LIN {X 0,Y 404.214,Z 398.218,A -85,B 0,C 180,E1 -10998.599,E2 -10998.599} C_VEL
LIN {X 0,Y 404.141,Z 398.144,A -85,B 0,C 180,E1 -11001.419,E2 -11001.419} C_VEL
LIN {X 0,Y 404.175,Z 398.142,A -85,B 0,C 180,E1 -11004.666,E2 -11004.666} C_VEL
LIN {X 0,Y 404.133,Z 398.136,A -85,B 0,C 180,E1 -11008.005,E2 -11008.005} C_VEL
LIN {X 0,Y 404.147,Z 398.137,A -85,B 0,C 180,E1 -11010.285,E2 -11010.285} C_VEL
LIN {X 0,Y 404.146,Z 398.13,A -85,B 0,C 180,E1 -11013.812,E2 -11013.812} C_VEL
LIN {X 0,Y 404.138,Z 398.142,A -85,B 0,C 180,E1 -11016.875,E2 -11016.875} C_VEL
LIN {X 0,Y 404.149,Z 398.142,A -85,B 0,C 180,E1 -11020.08,E2 -11020.08} C_VEL
LIN {X 0,Y 404.152,Z 398.144,A -85,B 0,C 180,E1 -11023.083,E2 -11023.083} C_VEL
LIN {X 0,Y 404.149,Z 398.138,A -85,B 0,C 180,E1 -11025.926,E2 -11025.926} C_VEL
LIN {X 0,Y 404.115,Z 398.146,A -85,B 0,C 180,E1 -11028.634,E2 -11028.634} C_VEL
LIN {X 0,Y 404.143,Z 398.126,A -85,B 0,C 180,E1 -11031.495,E2 -11031.495} C_VEL
LIN {X 0,Y 404.186,Z 398.126,A -85,B 0,C 180,E1 -11034.984,E2 -11034.984} C_VEL
LIN {X 0,Y 404.205,Z 398.311,A -85,B 0,C 180,E1 -11037.017,E2 -11037.017} C_VEL
LIN {X 0,Y 408.291,Z 414.179,A -85,B 0,C 180,E1 -11039.741,E2 -11039.741} C_VEL
LIN {X 0,Y 410.43,Z 423.971,A -85,B 0,C 180,E1 -11041.35,E2 -11041.35} C_VEL
LIN {X 0,Y 409.654,Z 440.641,A -85,B 0,C 180,E1 -11043.783,E2 -11043.783} C_VEL
LIN {X 0,Y 408.396,Z 462.743,A -85,B 0,C 180,E1 -11046.952,E2 -11046.952} C_VEL
LIN {X 0,Y 407.404,Z 484.784,A -85,B 0,C 180,E1 -11049.962,E2 -11049.962} C_VEL
LIN {X 0,Y 407.308,Z 487.804,A -85,B 0,C 180,E1 -11050.352,E2 -11050.352} C_VEL
LIN {X 0,Y 410.444,Z 509.789,A -85,B 0,C 180,E1 -11050.926,E2 -11050.926} C_VEL
LIN {X 0,Y 409.306,Z 600.036,A -85,B 0,C 180,E1 -11052.546,E2 -11052.546} C_VEL
LIN {X 0,Y 408.805,Z 613.109,A -85,B 0,C 180,E1 -11052.975,E2 -11052.975} C_VEL
LIN {X 0,Y 408.172,Z 626.084,A -85,B 0,C 180,E1 -11053.623,E2 -11053.623} C_VEL
LIN {X 0,Y 407.355,Z 638.791,A -85,B 0,C 180,E1 -11054.489,E2 -11054.489} C_VEL
LIN {X 0,Y 407.145,Z 642.093,A -85,B 0,C 180,E1 -11054.761,E2 -11054.761} C_VEL
LIN {X 0,Y 406.21,Z 647.1,A -85,B 0,C 180,E1 -11055.184,E2 -11055.184} C_VEL
LIN {X 0,Y 402.866,Z 654.993,A -85,B 0,C 180,E1 -11055.892,E2 -11055.892} C_VEL
LIN {X 0,Y 399.431,Z 662.416,A -85,B 0,C 180,E1 -11056.697,E2 -11056.697} C_VEL
LIN {X 0,Y 398.364,Z 666.666,A -85,B 0,C 180,E1 -11057.267,E2 -11057.267} C_VEL
LIN {X 0,Y 397.512,Z 676.011,A -85,B 0,C 180,E1 -11058.786,E2 -11058.786} C_VEL
LIN {X 0,Y 396.894,Z 683.473,A -85,B 0,C 180,E1 -11060.316,E2 -11060.316} C_VEL
LIN {X 0,Y 396.405,Z 689.464,A -85,B 0,C 180,E1 -11061.846,E2 -11061.846} C_VEL
LIN {X 0,Y 396.121,Z 694.52,A -85,B 0,C 180,E1 -11063.493,E2 -11063.493} C_VEL
LIN {X 0,Y 395.956,Z 697.833,A -85,B 0,C 180,E1 -11064.909,E2 -11064.909} C_VEL
LIN {X 0,Y 395.809,Z 699.703,A -85,B 0,C 180,E1 -11065.927,E2 -11065.927} C_VEL
LIN {X 0,Y 395.742,Z 701.131,A -85,B 0,C 180,E1 -11066.946,E2 -11066.946} C_VEL
LIN {X 0,Y 395.764,Z 702.132,A -85,B 0,C 180,E1 -11067.965,E2 -11067.965} C_VEL
LIN {X 0,Y 395.76,Z 702.986,A -85,B 0,C 180,E1 -11070,E2 -11070} C_VEL
LIN {X 0,Y 395.76,Z 702.794,A -85,B 0,C 180,E1 -11071.018,E2 -11071.018} C_VEL
LIN {X 0,Y 395.764,Z 702.205,A -85,B 0,C 180,E1 -11072.036,E2 -11072.036} C_VEL
LIN {X 0,Y 395.808,Z 699.863,A -85,B 0,C 180,E1 -11074.073,E2 -11074.073} C_VEL
LIN {X 0,Y 395.992,Z 696.979,A -85,B 0,C 180,E1 -11075.602,E2 -11075.602} C_VEL
LIN {X 0,Y 396.133,Z 693.063,A -85,B 0,C 180,E1 -11077.134,E2 -11077.134} C_VEL
LIN {X 0,Y 396.528,Z 687.99,A -85,B 0,C 180,E1 -11078.665,E2 -11078.665} C_VEL
LIN {X 0,Y 397.018,Z 681.596,A -85,B 0,C 180,E1 -11080.196,E2 -11080.196} C_VEL
LIN {X 0,Y 397.716,Z 673.654,A -85,B 0,C 180,E1 -11081.725,E2 -11081.725} C_VEL
LIN {X 0,Y 398.485,Z 665.541,A -85,B 0,C 180,E1 -11082.995,E2 -11082.995} C_VEL
LIN {X 0,Y 399.348,Z 655.573,A -85,B 0,C 180,E1 -11084.264,E2 -11084.264} C_VEL
LIN {X 0,Y 400.006,Z 645.746,A -85,B 0,C 180,E1 -11085.281,E2 -11085.281} C_VEL
LIN {X 0,Y 400.808,Z 635.099,A -85,B 0,C 180,E1 -11086.163,E2 -11086.163} C_VEL
LIN {X 0,Y 401.56,Z 623.437,A -85,B 0,C 180,E1 -11086.916,E2 -11086.916} C_VEL
LIN {X 0,Y 402.197,Z 610.726,A -85,B 0,C 180,E1 -11087.511,E2 -11087.511} C_VEL
LIN {X 0,Y 402.613,Z 597.392,A -85,B 0,C 180,E1 -11087.919,E2 -11087.919} C_VEL
LIN {X 0,Y 403.64,Z 509.348,A -85,B 0,C 180,E1 -11089.513,E2 -11089.513} C_VEL
LIN {X 0,Y 400.563,Z 487.69,A -85,B 0,C 180,E1 -11090.101,E2 -11090.101} C_VEL
LIN {X 0,Y 401.538,Z 465.188,A -85,B 0,C 180,E1 -11093.192,E2 -11093.192} C_VEL
LIN {X 0,Y 403.073,Z 439.157,A -85,B 0,C 180,E1 -11096.958,E2 -11096.958} C_VEL
LIN {X 0,Y 403.764,Z 426.144,A -85,B 0,C 180,E1 -11098.883,E2 -11098.883} C_VEL
LIN {X 0,Y 400.633,Z 412.28,A -85,B 0,C 180,E1 -11101.2,E2 -11101.2} C_VEL
LIN {X 0,Y 397.148,Z 399.203,A -85,B 0,C 180,E1 -11103.492,E2 -11103.492} C_VEL
LIN {X 0,Y 397.096,Z 399.012,A -85,B 0,C 180,E1 -11106.996,E2 -11106.996} C_VEL
LIN {X 0,Y 397.057,Z 399.012,A -85,B 0,C 180,E1 -11110.438,E2 -11110.438} C_VEL
LIN {X 0,Y 397.089,Z 399.01,A -85,B 0,C 180,E1 -11113.651,E2 -11113.651} C_VEL
LIN {X 0,Y 397.101,Z 399.019,A -85,B 0,C 180,E1 -11116.522,E2 -11116.522} C_VEL
LIN {X 0,Y 397.088,Z 399.022,A -85,B 0,C 180,E1 -11120.42,E2 -11120.42} C_VEL
LIN {X 0,Y 397.097,Z 399.012,A -85,B 0,C 180,E1 -11123.005,E2 -11123.005} C_VEL
LIN {X 0,Y 397.115,Z 399.006,A -85,B 0,C 180,E1 -11126.727,E2 -11126.727} C_VEL
LIN {X 0,Y 397.12,Z 399.011,A -85,B 0,C 180,E1 -11130.295,E2 -11130.295} C_VEL
LIN {X 0,Y 397.08,Z 399.027,A -85,B 0,C 180,E1 -11133.738,E2 -11133.738} C_VEL
LIN {X 0,Y 397.102,Z 399.008,A -85,B 0,C 180,E1 -11137.085,E2 -11137.085} C_VEL
LIN {X 0,Y 397.149,Z 399.009,A -85,B 0,C 180,E1 -11140.353,E2 -11140.353} C_VEL
LIN {X 0,Y 397.132,Z 399.008,A -85,B 0,C 180,E1 -11143.552,E2 -11143.552} C_VEL
LIN {X 0,Y 397.233,Z 398.998,A -85,B 0,C 180,E1 -11146.703,E2 -11146.703} C_VEL
LIN {X 0,Y 397.209,Z 398.996,A -85,B 0,C 180,E1 -11149.809,E2 -11149.809} C_VEL
LIN {X 0,Y 397.297,Z 398.992,A -85,B 0,C 180,E1 -11152.887,E2 -11152.887} C_VEL
LIN {X 0,Y 397.231,Z 398.989,A -85,B 0,C 180,E1 -11154.925,E2 -11154.925} C_VEL
LIN {X 0,Y 397.443,Z 398.978,A -85,B 0,C 180,E1 -11157.973,E2 -11157.973} C_VEL
LIN {X 0,Y 397.442,Z 398.959,A -85,B 0,C 180,E1 -11162.027,E2 -11162.027} C_VEL
LIN {X 0,Y 397.331,Z 398.992,A -85,B 0,C 180,E1 -11166.092,E2 -11166.092} C_VEL
LIN {X 0,Y 397.23,Z 398.989,A -85,B 0,C 180,E1 -11169.162,E2 -11169.162} C_VEL
LIN {X 0,Y 397.217,Z 399.005,A -85,B 0,C 180,E1 -11172.258,E2 -11172.258} C_VEL
LIN {X 0,Y 397.113,Z 399.01,A -85,B 0,C 180,E1 -11175.395,E2 -11175.395} C_VEL
LIN {X 0,Y 397.084,Z 399.018,A -85,B 0,C 180,E1 -11178.577,E2 -11178.577} C_VEL
LIN {X 0,Y 397.091,Z 399.012,A -85,B 0,C 180,E1 -11181.819,E2 -11181.819} C_VEL
LIN {X 0,Y 397.104,Z 399.015,A -85,B 0,C 180,E1 -11185.135,E2 -11185.135} C_VEL
LIN {X 0,Y 397.064,Z 399.01,A -85,B 0,C 180,E1 -11188.548,E2 -11188.548} C_VEL
LIN {X 0,Y 397.083,Z 399.026,A -85,B 0,C 180,E1 -11191.836,E2 -11191.836} C_VEL
LIN {X 0,Y 397.119,Z 399.007,A -85,B 0,C 180,E1 -11194.494,E2 -11194.494} C_VEL
LIN {X 0,Y 397.088,Z 399.015,A -85,B 0,C 180,E1 -11198.277,E2 -11198.277} C_VEL
LIN {X 0,Y 397.051,Z 398.989,A -85,B 0,C 180,E1 -11201.976,E2 -11201.976} C_VEL
LIN {X 0,Y 397.085,Z 399.02,A -85,B 0,C 180,E1 -11205.069,E2 -11205.069} C_VEL
LIN {X 0,Y 397.051,Z 398.999,A -85,B 0,C 180,E1 -11208.024,E2 -11208.024} C_VEL
LIN {X 0,Y 397.089,Z 399.017,A -85,B 0,C 180,E1 -11211.146,E2 -11211.146} C_VEL
LIN {X 0,Y 397.098,Z 399.022,A -85,B 0,C 180,E1 -11214.501,E2 -11214.501} C_VEL
LIN {X 0,Y 397.186,Z 399.276,A -85,B 0,C 180,E1 -11216.827,E2 -11216.827} C_VEL
LIN {X 0,Y 401.583,Z 418.852,A -85,B 0,C 180,E1 -11220.37,E2 -11220.37} C_VEL
LIN {X 0,Y 402.413,Z 422.758,A -85,B 0,C 180,E1 -11221.052,E2 -11221.052} C_VEL
LIN {X 0,Y 401.237,Z 439.938,A -85,B 0,C 180,E1 -11223.795,E2 -11223.795} C_VEL
LIN {X 0,Y 399.68,Z 461.77,A -85,B 0,C 180,E1 -11227.241,E2 -11227.241} C_VEL
LIN {X 0,Y 398.867,Z 475.69,A -85,B 0,C 180,E1 -11229.399,E2 -11229.399} C_VEL
LIN {X 0,Y 399.784,Z 488.481,A -85,B 0,C 180,E1 -11230.077,E2 -11230.077} C_VEL
LIN {X 0,Y 403.137,Z 518.848,A -85,B 0,C 180,E1 -11230.811,E2 -11230.811} C_VEL
LIN {X 0,Y 402.076,Z 606.296,A -85,B 0,C 180,E1 -11232.385,E2 -11232.385} C_VEL
LIN {X 0,Y 401.5,Z 619.645,A -85,B 0,C 180,E1 -11232.819,E2 -11232.819} C_VEL
LIN {X 0,Y 400.956,Z 632.32,A -85,B 0,C 180,E1 -11233.451,E2 -11233.451} C_VEL
LIN {X 0,Y 400.243,Z 643.58,A -85,B 0,C 180,E1 -11234.206,E2 -11234.206} C_VEL
LIN {X 0,Y 399.446,Z 654.245,A -85,B 0,C 180,E1 -11235.128,E2 -11235.128} C_VEL
LIN {X 0,Y 398.711,Z 664.528,A -85,B 0,C 180,E1 -11236.242,E2 -11236.242} C_VEL
LIN {X 0,Y 397.975,Z 673.995,A -85,B 0,C 180,E1 -11237.506,E2 -11237.506} C_VEL
LIN {X 0,Y 397.237,Z 681.776,A -85,B 0,C 180,E1 -11238.778,E2 -11238.778} C_VEL
LIN {X 0,Y 396.694,Z 689.349,A -85,B 0,C 180,E1 -11240.31,E2 -11240.31} C_VEL
LIN {X 0,Y 396.282,Z 695.425,A -85,B 0,C 180,E1 -11241.843,E2 -11241.843} C_VEL
LIN {X 0,Y 396.022,Z 700.221,A -85,B 0,C 180,E1 -11243.376,E2 -11243.376} C_VEL
LIN {X 0,Y 395.955,Z 703.879,A -85,B 0,C 180,E1 -11244.908,E2 -11244.908} C_VEL
LIN {X 0,Y 395.846,Z 705.763,A -85,B 0,C 180,E1 -11245.927,E2 -11245.927} C_VEL
LIN {X 0,Y 395.804,Z 707.185,A -85,B 0,C 180,E1 -11246.946,E2 -11246.946} C_VEL
LIN {X 0,Y 395.844,Z 708.188,A -85,B 0,C 180,E1 -11247.965,E2 -11247.965} C_VEL
LIN {X 0,Y 395.832,Z 708.801,A -85,B 0,C 180,E1 -11248.983,E2 -11248.983} C_VEL
LIN {X 0,Y 395.828,Z 709.02,A -85,B 0,C 180,E1 -11250,E2 -11250} C_VEL
LIN {X 0,Y 395.857,Z 708.799,A -85,B 0,C 180,E1 -11251.017,E2 -11251.017} C_VEL
LIN {X 0,Y 395.848,Z 708.184,A -85,B 0,C 180,E1 -11252.035,E2 -11252.035} C_VEL
LIN {X 0,Y 395.811,Z 707.18,A -85,B 0,C 180,E1 -11253.053,E2 -11253.053} C_VEL
LIN {X 0,Y 395.855,Z 705.755,A -85,B 0,C 180,E1 -11254.072,E2 -11254.072} C_VEL
LIN {X 0,Y 395.967,Z 702.789,A -85,B 0,C 180,E1 -11255.602,E2 -11255.602} C_VEL
LIN {X 0,Y 396.102,Z 698.758,A -85,B 0,C 180,E1 -11257.134,E2 -11257.134} C_VEL
LIN {X 0,Y 396.525,Z 692.538,A -85,B 0,C 180,E1 -11258.922,E2 -11258.922} C_VEL
LIN {X 0,Y 396.98,Z 685.747,A -85,B 0,C 180,E1 -11260.455,E2 -11260.455} C_VEL
LIN {X 0,Y 397.539,Z 678.792,A -85,B 0,C 180,E1 -11261.73,E2 -11261.73} C_VEL
LIN {X 0,Y 398.233,Z 670.382,A -85,B 0,C 180,E1 -11263.003,E2 -11263.003} C_VEL
LIN {X 0,Y 399.039,Z 659.963,A -85,B 0,C 180,E1 -11264.275,E2 -11264.275} C_VEL
LIN {X 0,Y 399.789,Z 649.629,A -85,B 0,C 180,E1 -11265.289,E2 -11265.289} C_VEL
LIN {X 0,Y 400.544,Z 638.228,A -85,B 0,C 180,E1 -11266.173,E2 -11266.173} C_VEL
LIN {X 0,Y 401.28,Z 626.381,A -85,B 0,C 180,E1 -11266.862,E2 -11266.862} C_VEL
LIN {X 0,Y 401.815,Z 613.578,A -85,B 0,C 180,E1 -11267.396,E2 -11267.396} C_VEL
LIN {X 0,Y 402.155,Z 599.896,A -85,B 0,C 180,E1 -11267.742,E2 -11267.742} C_VEL
LIN {X 0,Y 402.409,Z 587.532,A -85,B 0,C 180,E1 -11267.993,E2 -11267.993} C_VEL
LIN {X 0,Y 403.421,Z 551.708,A -85,B 0,C 180,E1 -11268.867,E2 -11268.867} C_VEL
LIN {X 0,Y 404.277,Z 517.801,A -85,B 0,C 180,E1 -11269.699,E2 -11269.699} C_VEL
LIN {X 0,Y 402.318,Z 492.103,A -85,B 0,C 180,E1 -11270.547,E2 -11270.547} C_VEL
LIN {X 0,Y 399.514,Z 472.889,A -85,B 0,C 180,E1 -11271.317,E2 -11271.317} C_VEL
LIN {X 0,Y 399.185,Z 470.402,A -85,B 0,C 180,E1 -11271.458,E2 -11271.458} C_VEL
LIN {X 0,Y 400.855,Z 449.87,A -85,B 0,C 180,E1 -11274.884,E2 -11274.884} C_VEL
LIN {X 0,Y 402.767,Z 431.494,A -85,B 0,C 180,E1 -11278.108,E2 -11278.108} C_VEL
LIN {X 0,Y 403.442,Z 425.577,A -85,B 0,C 180,E1 -11279.194,E2 -11279.194} C_VEL
LIN {X 0,Y 402.201,Z 418.214,A -85,B 0,C 180,E1 -11280.782,E2 -11280.782} C_VEL
LIN {X 0,Y 399.687,Z 407.941,A -85,B 0,C 180,E1 -11283.271,E2 -11283.271} C_VEL
LIN {X 0,Y 397.125,Z 399.276,A -85,B 0,C 180,E1 -11285.733,E2 -11285.733} C_VEL
LIN {X 0,Y 397.087,Z 399.023,A -85,B 0,C 180,E1 -11287.207,E2 -11287.207} C_VEL
LIN {X 0,Y 397.055,Z 399.026,A -85,B 0,C 180,E1 -11290.437,E2 -11290.437} C_VEL
LIN {X 0,Y 397.087,Z 399.022,A -85,B 0,C 180,E1 -11293.651,E2 -11293.651} C_VEL
LIN {X 0,Y 397.092,Z 399.02,A -85,B 0,C 180,E1 -11296.523,E2 -11296.523} C_VEL
LIN {X 0,Y 397.087,Z 399.021,A -85,B 0,C 180,E1 -11300.419,E2 -11300.419} C_VEL
LIN {X 0,Y 397.096,Z 399.022,A -85,B 0,C 180,E1 -11303.005,E2 -11303.005} C_VEL
LIN {X 0,Y 397.12,Z 399.019,A -85,B 0,C 180,E1 -11306.282,E2 -11306.282} C_VEL
LIN {X 0,Y 397.102,Z 399.022,A -85,B 0,C 180,E1 -11310.137,E2 -11310.137} C_VEL
LIN {X 0,Y 397.097,Z 399.023,A -85,B 0,C 180,E1 -11313.739,E2 -11313.739} C_VEL
LIN {X 0,Y 397.11,Z 399.02,A -85,B 0,C 180,E1 -11317.086,E2 -11317.086} C_VEL
LIN {X 0,Y 397.146,Z 399.215,A -85,B 0,C 180,E1 -11318.716,E2 -11318.716} C_VEL
LIN {X 0,Y 397.321,Z 400.037,A -85,B 0,C 180,E1 -11318.883,E2 -11318.883} C_VEL
LIN {X 0,Y 403.54,Z 412.118,A -85,B 0,C 180,E1 -11319.838,E2 -11319.838} C_VEL
LIN {X 0,Y 406.442,Z 418.563,A -85,B 0,C 180,E1 -11320.273,E2 -11320.273} C_VEL
LIN {X 0,Y 404.512,Z 480.076,A -85,B 0,C 180,E1 -11321.842,E2 -11321.842} C_VEL
LIN {X 0,Y 404.373,Z 494.158,A -85,B 0,C 180,E1 -11322.293,E2 -11322.293} C_VEL
LIN {X 0,Y 404.15,Z 506.725,A -85,B 0,C 180,E1 -11322.904,E2 -11322.904} C_VEL
LIN {X 0,Y 403.667,Z 517.528,A -85,B 0,C 180,E1 -11323.591,E2 -11323.591} C_VEL
LIN {X 0,Y 402.996,Z 529.51,A -85,B 0,C 180,E1 -11324.577,E2 -11324.577} C_VEL
LIN {X 0,Y 402.285,Z 539.345,A -85,B 0,C 180,E1 -11325.585,E2 -11325.585} C_VEL
LIN {X 0,Y 401.52,Z 549.276,A -85,B 0,C 180,E1 -11326.847,E2 -11326.847} C_VEL
LIN {X 0,Y 400.62,Z 558.724,A -85,B 0,C 180,E1 -11328.361,E2 -11328.361} C_VEL
LIN {X 0,Y 399.882,Z 566.235,A -85,B 0,C 180,E1 -11329.878,E2 -11329.878} C_VEL
LIN {X 0,Y 399.211,Z 572.153,A -85,B 0,C 180,E1 -11331.394,E2 -11331.394} C_VEL
LIN {X 0,Y 398.562,Z 576.822,A -85,B 0,C 180,E1 -11332.91,E2 -11332.91} C_VEL
LIN {X 0,Y 398.232,Z 579.283,A -85,B 0,C 180,E1 -11333.922,E2 -11333.922} C_VEL
LIN {X 0,Y 398.021,Z 581.233,A -85,B 0,C 180,E1 -11334.935,E2 -11334.935} C_VEL
LIN {X 0,Y 397.88,Z 582.698,A -85,B 0,C 180,E1 -11335.948,E2 -11335.948} C_VEL
LIN {X 0,Y 397.671,Z 583.762,A -85,B 0,C 180,E1 -11336.961,E2 -11336.961} C_VEL
LIN {X 0,Y 397.521,Z 584.391,A -85,B 0,C 180,E1 -11337.974,E2 -11337.974} C_VEL
LIN {X 0,Y 397.32,Z 584.575,A -85,B 0,C 180,E1 -11338.987,E2 -11338.987} C_VEL
LIN {X 0,Y 397.209,Z 584.343,A -85,B 0,C 180,E1 -11340,E2 -11340} C_VEL
LIN {X 0,Y 397.214,Z 583.688,A -85,B 0,C 180,E1 -11341.014,E2 -11341.014} C_VEL
LIN {X 0,Y 397.139,Z 582.587,A -85,B 0,C 180,E1 -11342.028,E2 -11342.028} C_VEL
LIN {X 0,Y 397.267,Z 581.044,A -85,B 0,C 180,E1 -11343.042,E2 -11343.042} C_VEL
LIN {X 0,Y 397.261,Z 577.926,A -85,B 0,C 180,E1 -11344.566,E2 -11344.566} C_VEL
LIN {X 0,Y 397.516,Z 573.698,A -85,B 0,C 180,E1 -11346.089,E2 -11346.089} C_VEL
LIN {X 0,Y 397.898,Z 568.266,A -85,B 0,C 180,E1 -11347.612,E2 -11347.612} C_VEL
LIN {X 0,Y 398.132,Z 561.464,A -85,B 0,C 180,E1 -11349.142,E2 -11349.142} C_VEL
LIN {X 0,Y 398.562,Z 552.952,A -85,B 0,C 180,E1 -11350.67,E2 -11350.67} C_VEL
LIN {X 0,Y 398.96,Z 544.272,A -85,B 0,C 180,E1 -11351.946,E2 -11351.946} C_VEL
LIN {X 0,Y 399.4,Z 534.8,A -85,B 0,C 180,E1 -11353.094,E2 -11353.094} C_VEL
LIN {X 0,Y 399.983,Z 523.027,A -85,B 0,C 180,E1 -11354.24,E2 -11354.24} C_VEL
LIN {X 0,Y 400.331,Z 511.226,A -85,B 0,C 180,E1 -11355.16,E2 -11355.16} C_VEL
LIN {X 0,Y 400.673,Z 498.625,A -85,B 0,C 180,E1 -11355.907,E2 -11355.907} C_VEL
LIN {X 0,Y 400.911,Z 485.21,A -85,B 0,C 180,E1 -11356.485,E2 -11356.485} C_VEL
LIN {X 0,Y 400.964,Z 470.966,A -85,B 0,C 180,E1 -11356.876,E2 -11356.876} C_VEL
LIN {X 0,Y 401.898,Z 413.794,A -85,B 0,C 180,E1 -11358.138,E2 -11358.138} C_VEL
LIN {X 0,Y 397.351,Z 399.974,A -85,B 0,C 180,E1 -11358.64,E2 -11358.64} C_VEL
LIN {X 0,Y 397.179,Z 399.09,A -85,B 0,C 180,E1 -11358.84,E2 -11358.84} C_VEL
LIN {X 0,Y 397.1,Z 399.02,A -85,B 0,C 180,E1 -11361.818,E2 -11361.818} C_VEL
LIN {X 0,Y 397.132,Z 399.017,A -85,B 0,C 180,E1 -11365.133,E2 -11365.133} C_VEL
LIN {X 0,Y 397.081,Z 399.011,A -85,B 0,C 180,E1 -11368.547,E2 -11368.547} C_VEL
LIN {X 0,Y 397.084,Z 399.021,A -85,B 0,C 180,E1 -11371.837,E2 -11371.837} C_VEL
LIN {X 0,Y 397.127,Z 399.007,A -85,B 0,C 180,E1 -11374.493,E2 -11374.493} C_VEL
LIN {X 0,Y 397.102,Z 399.012,A -85,B 0,C 180,E1 -11378.275,E2 -11378.275} C_VEL
LIN {X 0,Y 397.088,Z 399.02,A -85,B 0,C 180,E1 -11380.909,E2 -11380.909} C_VEL
LIN {X 0,Y 397.102,Z 399.02,A -85,B 0,C 180,E1 -11383.649,E2 -11383.649} C_VEL
LIN {X 0,Y 397.103,Z 399.022,A -85,B 0,C 180,E1 -11386.521,E2 -11386.521} C_VEL
LIN {X 0,Y 397.102,Z 399.02,A -85,B 0,C 180,E1 -11389.555,E2 -11389.555} C_VEL
LIN {X 0,Y 397.099,Z 399.02,A -85,B 0,C 180,E1 -11393.005,E2 -11393.005} C_VEL
LIN {X 0,Y 397.164,Z 399.117,A -85,B 0,C 180,E1 -11396.565,E2 -11396.565} C_VEL
LIN {X 0,Y 397.56,Z 400.72,A -85,B 0,C 180,E1 -11396.917,E2 -11396.917} C_VEL
LIN {X 0,Y 401.476,Z 415.681,A -85,B 0,C 180,E1 -11399.492,E2 -11399.492} C_VEL
LIN {X 0,Y 403.559,Z 425.307,A -85,B 0,C 180,E1 -11401.101,E2 -11401.101} C_VEL
LIN {X 0,Y 403.51,Z 430.992,A -85,B 0,C 180,E1 -11401.949,E2 -11401.949} C_VEL
LIN {X 0,Y 402.287,Z 451.389,A -85,B 0,C 180,E1 -11404.935,E2 -11404.935} C_VEL
LIN {X 0,Y 400.98,Z 475.834,A -85,B 0,C 180,E1 -11408.404,E2 -11408.404} C_VEL
LIN {X 0,Y 400.488,Z 487.788,A -85,B 0,C 180,E1 -11410.003,E2 -11410.003} C_VEL
LIN {X 0,Y 403.668,Z 509.71,A -85,B 0,C 180,E1 -11410.593,E2 -11410.593} C_VEL
LIN {X 0,Y 402.93,Z 575.061,A -85,B 0,C 180,E1 -11411.768,E2 -11411.768} C_VEL
LIN {X 0,Y 402.55,Z 601.314,A -85,B 0,C 180,E1 -11412.276,E2 -11412.276} C_VEL
LIN {X 0,Y 401.964,Z 614.543,A -85,B 0,C 180,E1 -11412.741,E2 -11412.741} C_VEL
LIN {X 0,Y 401.271,Z 627.186,A -85,B 0,C 180,E1 -11413.399,E2 -11413.399} C_VEL
LIN {X 0,Y 400.533,Z 638.833,A -85,B 0,C 180,E1 -11414.218,E2 -11414.218} C_VEL
LIN {X 0,Y 399.693,Z 650.295,A -85,B 0,C 180,E1 -11415.262,E2 -11415.262} C_VEL
LIN {X 0,Y 398.882,Z 661.083,A -85,B 0,C 180,E1 -11416.5,E2 -11416.5} C_VEL
LIN {X 0,Y 398.364,Z 666.666,A -85,B 0,C 180,E1 -11417.267,E2 -11417.267} C_VEL
LIN {X 0,Y 397.318,Z 670.755,A -85,B 0,C 180,E1 -11417.867,E2 -11417.867} C_VEL
LIN {X 0,Y 393.943,Z 677.055,A -85,B 0,C 180,E1 -11418.864,E2 -11418.864} C_VEL
LIN {X 0,Y 390.632,Z 682.716,A -85,B 0,C 180,E1 -11419.95,E2 -11419.95} C_VEL
LIN {X 0,Y 389.699,Z 685.775,A -85,B 0,C 180,E1 -11420.679,E2 -11420.679} C_VEL
LIN {X 0,Y 389.236,Z 691.244,A -85,B 0,C 180,E1 -11422.217,E2 -11422.217} C_VEL
LIN {X 0,Y 388.963,Z 695.597,A -85,B 0,C 180,E1 -11423.776,E2 -11423.776} C_VEL
LIN {X 0,Y 388.88,Z 697.888,A -85,B 0,C 180,E1 -11424.816,E2 -11424.816} C_VEL
LIN {X 0,Y 388.738,Z 699.757,A -85,B 0,C 180,E1 -11425.853,E2 -11425.853} C_VEL
LIN {X 0,Y 388.65,Z 701.186,A -85,B 0,C 180,E1 -11426.89,E2 -11426.89} C_VEL
LIN {X 0,Y 388.662,Z 702.186,A -85,B 0,C 180,E1 -11427.928,E2 -11427.928} C_VEL
LIN {X 0,Y 388.673,Z 703.04,A -85,B 0,C 180,E1 -11430,E2 -11430} C_VEL
LIN {X 0,Y 388.659,Z 702.847,A -85,B 0,C 180,E1 -11431.036,E2 -11431.036} C_VEL
LIN {X 0,Y 388.662,Z 702.259,A -85,B 0,C 180,E1 -11432.073,E2 -11432.073} C_VEL
LIN {X 0,Y 388.736,Z 699.916,A -85,B 0,C 180,E1 -11434.147,E2 -11434.147} C_VEL
LIN {X 0,Y 388.897,Z 697.032,A -85,B 0,C 180,E1 -11435.704,E2 -11435.704} C_VEL
LIN {X 0,Y 389.085,Z 693.115,A -85,B 0,C 180,E1 -11437.264,E2 -11437.264} C_VEL
LIN {X 0,Y 389.505,Z 688.04,A -85,B 0,C 180,E1 -11438.822,E2 -11438.822} C_VEL
LIN {X 0,Y 390.011,Z 681.644,A -85,B 0,C 180,E1 -11440.382,E2 -11440.382} C_VEL
LIN {X 0,Y 390.752,Z 673.701,A -85,B 0,C 180,E1 -11441.937,E2 -11441.937} C_VEL
LIN {X 0,Y 391.56,Z 665.585,A -85,B 0,C 180,E1 -11443.229,E2 -11443.229} C_VEL
LIN {X 0,Y 392.446,Z 655.613,A -85,B 0,C 180,E1 -11444.52,E2 -11444.52} C_VEL
LIN {X 0,Y 393.149,Z 645.781,A -85,B 0,C 180,E1 -11445.554,E2 -11445.554} C_VEL
LIN {X 0,Y 394.008,Z 635.127,A -85,B 0,C 180,E1 -11446.449,E2 -11446.449} C_VEL
LIN {X 0,Y 394.763,Z 623.455,A -85,B 0,C 180,E1 -11447.216,E2 -11447.216} C_VEL
LIN {X 0,Y 395.444,Z 610.72,A -85,B 0,C 180,E1 -11447.82,E2 -11447.82} C_VEL
LIN {X 0,Y 395.88,Z 597.342,A -85,B 0,C 180,E1 -11448.234,E2 -11448.234} C_VEL
LIN {X 0,Y 397.016,Z 510.534,A -85,B 0,C 180,E1 -11449.828,E2 -11449.828} C_VEL
LIN {X 0,Y 393.757,Z 487.918,A -85,B 0,C 180,E1 -11450.445,E2 -11450.445} C_VEL
LIN {X 0,Y 394.58,Z 468.765,A -85,B 0,C 180,E1 -11453.07,E2 -11453.07} C_VEL
LIN {X 0,Y 396.183,Z 442.546,A -85,B 0,C 180,E1 -11456.895,E2 -11456.895} C_VEL
LIN {X 0,Y 396.999,Z 427.883,A -85,B 0,C 180,E1 -11459.086,E2 -11459.086} C_VEL
LIN {X 0,Y 393.806,Z 413.868,A -85,B 0,C 180,E1 -11461.467,E2 -11461.467} C_VEL
LIN {X 0,Y 390.103,Z 400.047,A -85,B 0,C 180,E1 -11463.932,E2 -11463.932} C_VEL
LIN {X 0,Y 390.056,Z 399.889,A -85,B 0,C 180,E1 -11466.484,E2 -11466.484} C_VEL
LIN {X 0,Y 390.038,Z 399.894,A -85,B 0,C 180,E1 -11469.212,E2 -11469.212} C_VEL
LIN {X 0,Y 390.032,Z 399.901,A -85,B 0,C 180,E1 -11472.372,E2 -11472.372} C_VEL
LIN {X 0,Y 390.045,Z 399.879,A -85,B 0,C 180,E1 -11475.354,E2 -11475.354} C_VEL
LIN {X 0,Y 390.019,Z 399.903,A -85,B 0,C 180,E1 -11478.185,E2 -11478.185} C_VEL
LIN {X 0,Y 390.06,Z 399.898,A -85,B 0,C 180,E1 -11480.904,E2 -11480.904} C_VEL
LIN {X 0,Y 390.072,Z 399.894,A -85,B 0,C 180,E1 -11484.792,E2 -11484.792} C_VEL
LIN {X 0,Y 390.026,Z 399.901,A -85,B 0,C 180,E1 -11488.496,E2 -11488.496} C_VEL
LIN {X 0,Y 390.018,Z 399.897,A -85,B 0,C 180,E1 -11492.003,E2 -11492.003} C_VEL
LIN {X 0,Y 390.046,Z 399.892,A -85,B 0,C 180,E1 -11495.517,E2 -11495.517} C_VEL
LIN {X 0,Y 390.065,Z 399.895,A -85,B 0,C 180,E1 -11498.878,E2 -11498.878} C_VEL
LIN {X 0,Y 390.072,Z 399.881,A -85,B 0,C 180,E1 -11502.164,E2 -11502.164} C_VEL
LIN {X 0,Y 390.096,Z 399.893,A -85,B 0,C 180,E1 -11505.391,E2 -11505.391} C_VEL
LIN {X 0,Y 390.171,Z 399.872,A -85,B 0,C 180,E1 -11507.517,E2 -11507.517} C_VEL
LIN {X 0,Y 390.189,Z 399.876,A -85,B 0,C 180,E1 -11510.671,E2 -11510.671} C_VEL
LIN {X 0,Y 390.279,Z 399.861,A -85,B 0,C 180,E1 -11513.797,E2 -11513.797} C_VEL
LIN {X 0,Y 390.41,Z 399.853,A -85,B 0,C 180,E1 -11517.937,E2 -11517.937} C_VEL
LIN {X 0,Y 390.408,Z 399.834,A -85,B 0,C 180,E1 -11522.063,E2 -11522.063} C_VEL
LIN {X 0,Y 390.286,Z 399.869,A -85,B 0,C 180,E1 -11526.203,E2 -11526.203} C_VEL
LIN {X 0,Y 390.189,Z 399.865,A -85,B 0,C 180,E1 -11529.329,E2 -11529.329} C_VEL
LIN {X 0,Y 390.17,Z 399.881,A -85,B 0,C 180,E1 -11532.483,E2 -11532.483} C_VEL
LIN {X 0,Y 390.056,Z 399.884,A -85,B 0,C 180,E1 -11535.68,E2 -11535.68} C_VEL
LIN {X 0,Y 390.042,Z 399.895,A -85,B 0,C 180,E1 -11538.925,E2 -11538.925} C_VEL
LIN {X 0,Y 390.033,Z 399.886,A -85,B 0,C 180,E1 -11542.235,E2 -11542.235} C_VEL
LIN {X 0,Y 390.053,Z 399.899,A -85,B 0,C 180,E1 -11545.722,E2 -11545.722} C_VEL
LIN {X 0,Y 390.026,Z 399.886,A -85,B 0,C 180,E1 -11549.112,E2 -11549.112} C_VEL
LIN {X 0,Y 390.044,Z 399.895,A -85,B 0,C 180,E1 -11552.721,E2 -11552.721} C_VEL
LIN {X 0,Y 390.044,Z 399.895,A -85,B 0,C 180,E1 -11555.822,E2 -11555.822} C_VEL
LIN {X 0,Y 390.035,Z 399.885,A -85,B 0,C 180,E1 -11559.211,E2 -11559.211} C_VEL
LIN {X 0,Y 390.03,Z 399.867,A -85,B 0,C 180,E1 -11562.371,E2 -11562.371} C_VEL
LIN {X 0,Y 390.041,Z 399.899,A -85,B 0,C 180,E1 -11565.353,E2 -11565.353} C_VEL
LIN {X 0,Y 390.015,Z 399.873,A -85,B 0,C 180,E1 -11568.184,E2 -11568.184} C_VEL
LIN {X 0,Y 390.055,Z 399.893,A -85,B 0,C 180,E1 -11570.903,E2 -11570.903} C_VEL
LIN {X 0,Y 390.069,Z 399.898,A -85,B 0,C 180,E1 -11574.791,E2 -11574.791} C_VEL
LIN {X 0,Y 390.113,Z 400.1,A -85,B 0,C 180,E1 -11576.553,E2 -11576.553} C_VEL
LIN {X 0,Y 394.416,Z 419.179,A -85,B 0,C 180,E1 -11580.071,E2 -11580.071} C_VEL
LIN {X 0,Y 395.492,Z 425.129,A -85,B 0,C 180,E1 -11581.12,E2 -11581.12} C_VEL
LIN {X 0,Y 393.889,Z 445.14,A -85,B 0,C 180,E1 -11584.362,E2 -11584.362} C_VEL
LIN {X 0,Y 392.521,Z 463.799,A -85,B 0,C 180,E1 -11587.359,E2 -11587.359} C_VEL
LIN {X 0,Y 391.959,Z 473.749,A -85,B 0,C 180,E1 -11588.92,E2 -11588.92} C_VEL
LIN {X 0,Y 393.054,Z 488.867,A -85,B 0,C 180,E1 -11589.727,E2 -11589.727} C_VEL
LIN {X 0,Y 396.47,Z 519.831,A -85,B 0,C 180,E1 -11590.492,E2 -11590.492} C_VEL
LIN {X 0,Y 395.341,Z 606.342,A -85,B 0,C 180,E1 -11592.075,E2 -11592.075} C_VEL
LIN {X 0,Y 394.744,Z 619.641,A -85,B 0,C 180,E1 -11592.516,E2 -11592.516} C_VEL
LIN {X 0,Y 394.165,Z 632.299,A -85,B 0,C 180,E1 -11593.157,E2 -11593.157} C_VEL
LIN {X 0,Y 393.408,Z 643.548,A -85,B 0,C 180,E1 -11593.925,E2 -11593.925} C_VEL
LIN {X 0,Y 392.581,Z 654.208,A -85,B 0,C 180,E1 -11594.862,E2 -11594.862} C_VEL
LIN {X 0,Y 391.751,Z 664.894,A -85,B 0,C 180,E1 -11596.043,E2 -11596.043} C_VEL
LIN {X 0,Y 391.024,Z 673.95,A -85,B 0,C 180,E1 -11597.281,E2 -11597.281} C_VEL
LIN {X 0,Y 390.254,Z 681.729,A -85,B 0,C 180,E1 -11598.574,E2 -11598.574} C_VEL
LIN {X 0,Y 389.683,Z 689.3,A -85,B 0,C 180,E1 -11600.134,E2 -11600.134} C_VEL
LIN {X 0,Y 389.237,Z 695.374,A -85,B 0,C 180,E1 -11601.695,E2 -11601.695} C_VEL
LIN {X 0,Y 388.954,Z 700.169,A -85,B 0,C 180,E1 -11603.255,E2 -11603.255} C_VEL
LIN {X 0,Y 388.87,Z 703.827,A -85,B 0,C 180,E1 -11604.815,E2 -11604.815} C_VEL
LIN {X 0,Y 388.77,Z 705.71,A -85,B 0,C 180,E1 -11605.853,E2 -11605.853} C_VEL
LIN {X 0,Y 388.708,Z 707.132,A -85,B 0,C 180,E1 -11606.891,E2 -11606.891} C_VEL
LIN {X 0,Y 388.741,Z 708.134,A -85,B 0,C 180,E1 -11607.928,E2 -11607.928} C_VEL
LIN {X 0,Y 388.744,Z 708.747,A -85,B 0,C 180,E1 -11608.964,E2 -11608.964} C_VEL
LIN {X 0,Y 388.755,Z 708.966,A -85,B 0,C 180,E1 -11610,E2 -11610} C_VEL
LIN {X 0,Y 388.784,Z 708.745,A -85,B 0,C 180,E1 -11611.036,E2 -11611.036} C_VEL
LIN {X 0,Y 388.745,Z 708.13,A -85,B 0,C 180,E1 -11612.072,E2 -11612.072} C_VEL
LIN {X 0,Y 388.715,Z 707.126,A -85,B 0,C 180,E1 -11613.109,E2 -11613.109} C_VEL
LIN {X 0,Y 388.78,Z 705.701,A -85,B 0,C 180,E1 -11614.146,E2 -11614.146} C_VEL
LIN {X 0,Y 388.875,Z 702.12,A -85,B 0,C 180,E1 -11615.963,E2 -11615.963} C_VEL
LIN {X 0,Y 389.112,Z 697.096,A -85,B 0,C 180,E1 -11617.785,E2 -11617.785} C_VEL
LIN {X 0,Y 389.565,Z 691.48,A -85,B 0,C 180,E1 -11619.344,E2 -11619.344} C_VEL
LIN {X 0,Y 390.068,Z 684.403,A -85,B 0,C 180,E1 -11620.905,E2 -11620.905} C_VEL
LIN {X 0,Y 390.837,Z 675.556,A -85,B 0,C 180,E1 -11622.461,E2 -11622.461} C_VEL
LIN {X 0,Y 391.631,Z 666.686,A -85,B 0,C 180,E1 -11623.724,E2 -11623.724} C_VEL
LIN {X 0,Y 392.366,Z 656.694,A -85,B 0,C 180,E1 -11624.881,E2 -11624.881} C_VEL
LIN {X 0,Y 393.247,Z 645.028,A -85,B 0,C 180,E1 -11625.949,E2 -11625.949} C_VEL
LIN {X 0,Y 394.084,Z 633.261,A -85,B 0,C 180,E1 -11626.779,E2 -11626.779} C_VEL
LIN {X 0,Y 394.775,Z 620.204,A -85,B 0,C 180,E1 -11627.449,E2 -11627.449} C_VEL
LIN {X 0,Y 395.273,Z 607.259,A -85,B 0,C 180,E1 -11627.894,E2 -11627.894} C_VEL
LIN {X 0,Y 395.586,Z 590.959,A -85,B 0,C 180,E1 -11628.248,E2 -11628.248} C_VEL
LIN {X 0,Y 396.206,Z 576.323,A -85,B 0,C 180,E1 -11628.687,E2 -11628.687} C_VEL
LIN {X 0,Y 397.953,Z 519.392,A -85,B 0,C 180,E1 -11630.093,E2 -11630.093} C_VEL
LIN {X 0,Y 396.054,Z 493.38,A -85,B 0,C 180,E1 -11630.982,E2 -11630.982} C_VEL
LIN {X 0,Y 393.263,Z 474.029,A -85,B 0,C 180,E1 -11631.792,E2 -11631.792} C_VEL
LIN {X 0,Y 392.466,Z 468.95,A -85,B 0,C 180,E1 -11632.054,E2 -11632.054} C_VEL
LIN {X 0,Y 394.006,Z 451.322,A -85,B 0,C 180,E1 -11635.064,E2 -11635.064} C_VEL
LIN {X 0,Y 396.065,Z 433.149,A -85,B 0,C 180,E1 -11638.338,E2 -11638.338} C_VEL
LIN {X 0,Y 396.738,Z 427.054,A -85,B 0,C 180,E1 -11639.486,E2 -11639.486} C_VEL
LIN {X 0,Y 395.2,Z 418.639,A -85,B 0,C 180,E1 -11641.394,E2 -11641.394} C_VEL
LIN {X 0,Y 392.954,Z 409.75,A -85,B 0,C 180,E1 -11643.672,E2 -11643.672} C_VEL
LIN {X 0,Y 390.646,Z 402.017,A -85,B 0,C 180,E1 -11645.945,E2 -11645.945} C_VEL
LIN {X 0,Y 390.061,Z 399.979,A -85,B 0,C 180,E1 -11646.644,E2 -11646.644} C_VEL
LIN {X 0,Y 390.036,Z 399.902,A -85,B 0,C 180,E1 -11649.212,E2 -11649.212} C_VEL
LIN {X 0,Y 390.03,Z 399.902,A -85,B 0,C 180,E1 -11652.372,E2 -11652.372} C_VEL
LIN {X 0,Y 390.041,Z 399.899,A -85,B 0,C 180,E1 -11655.354,E2 -11655.354} C_VEL
LIN {X 0,Y 390.015,Z 399.902,A -85,B 0,C 180,E1 -11658.184,E2 -11658.184} C_VEL
LIN {X 0,Y 390.058,Z 399.898,A -85,B 0,C 180,E1 -11660.904,E2 -11660.904} C_VEL
LIN {X 0,Y 390.085,Z 399.895,A -85,B 0,C 180,E1 -11664.793,E2 -11664.793} C_VEL
LIN {X 0,Y 390.025,Z 399.903,A -85,B 0,C 180,E1 -11668.496,E2 -11668.496} C_VEL
LIN {X 0,Y 390.041,Z 399.901,A -85,B 0,C 180,E1 -11672.064,E2 -11672.064} C_VEL
LIN {X 0,Y 390.065,Z 399.898,A -85,B 0,C 180,E1 -11675.518,E2 -11675.518} C_VEL
LIN {X 0,Y 390.071,Z 400.021,A -85,B 0,C 180,E1 -11677.998,E2 -11677.998} C_VEL
LIN {X 0,Y 390.253,Z 400.849,A -85,B 0,C 180,E1 -11678.204,E2 -11678.204} C_VEL
LIN {X 0,Y 391.746,Z 403.695,A -85,B 0,C 180,E1 -11678.475,E2 -11678.475} C_VEL
LIN {X 0,Y 398.316,Z 416.462,A -85,B 0,C 180,E1 -11679.522,E2 -11679.522} C_VEL
LIN {X 0,Y 400.279,Z 420.705,A -85,B 0,C 180,E1 -11679.82,E2 -11679.82} C_VEL
LIN {X 0,Y 398.141,Z 480.891,A -85,B 0,C 180,E1 -11681.412,E2 -11681.412} C_VEL
LIN {X 0,Y 397.987,Z 494.92,A -85,B 0,C 180,E1 -11681.866,E2 -11681.866} C_VEL
LIN {X 0,Y 397.706,Z 508.156,A -85,B 0,C 180,E1 -11682.518,E2 -11682.518} C_VEL
LIN {X 0,Y 397.177,Z 519.98,A -85,B 0,C 180,E1 -11683.297,E2 -11683.297} C_VEL
LIN {X 0,Y 396.421,Z 531.838,A -85,B 0,C 180,E1 -11684.314,E2 -11684.314} C_VEL
LIN {X 0,Y 395.675,Z 541.407,A -85,B 0,C 180,E1 -11685.338,E2 -11685.338} C_VEL
LIN {X 0,Y 394.821,Z 551.089,A -85,B 0,C 180,E1 -11686.62,E2 -11686.62} C_VEL
LIN {X 0,Y 393.88,Z 560.448,A -85,B 0,C 180,E1 -11688.159,E2 -11688.159} C_VEL
LIN {X 0,Y 393.074,Z 567.837,A -85,B 0,C 180,E1 -11689.7,E2 -11689.7} C_VEL
LIN {X 0,Y 392.37,Z 573.673,A -85,B 0,C 180,E1 -11691.243,E2 -11691.243} C_VEL
LIN {X 0,Y 391.67,Z 578.236,A -85,B 0,C 180,E1 -11692.784,E2 -11692.784} C_VEL
LIN {X 0,Y 391.311,Z 580.642,A -85,B 0,C 180,E1 -11693.814,E2 -11693.814} C_VEL
LIN {X 0,Y 391.068,Z 582.513,A -85,B 0,C 180,E1 -11694.845,E2 -11694.845} C_VEL
LIN {X 0,Y 390.923,Z 583.937,A -85,B 0,C 180,E1 -11695.876,E2 -11695.876} C_VEL
LIN {X 0,Y 390.694,Z 584.966,A -85,B 0,C 180,E1 -11696.907,E2 -11696.907} C_VEL
LIN {X 0,Y 390.525,Z 585.529,A -85,B 0,C 180,E1 -11697.937,E2 -11697.937} C_VEL
LIN {X 0,Y 390.324,Z 585.669,A -85,B 0,C 180,E1 -11698.968,E2 -11698.968} C_VEL
LIN {X 0,Y 390.188,Z 585.393,A -85,B 0,C 180,E1 -11700,E2 -11700} C_VEL
LIN {X 0,Y 390.189,Z 584.672,A -85,B 0,C 180,E1 -11701.032,E2 -11701.032} C_VEL
LIN {X 0,Y 390.116,Z 583.514,A -85,B 0,C 180,E1 -11702.065,E2 -11702.065} C_VEL
LIN {X 0,Y 390.156,Z 580.966,A -85,B 0,C 180,E1 -11703.615,E2 -11703.615} C_VEL
LIN {X 0,Y 390.28,Z 577.381,A -85,B 0,C 180,E1 -11705.166,E2 -11705.166} C_VEL
LIN {X 0,Y 390.583,Z 572.654,A -85,B 0,C 180,E1 -11706.717,E2 -11706.717} C_VEL
LIN {X 0,Y 390.918,Z 566.671,A -85,B 0,C 180,E1 -11708.269,E2 -11708.269} C_VEL
LIN {X 0,Y 391.265,Z 559.21,A -85,B 0,C 180,E1 -11709.825,E2 -11709.825} C_VEL
LIN {X 0,Y 391.801,Z 549.871,A -85,B 0,C 180,E1 -11711.38,E2 -11711.38} C_VEL
LIN {X 0,Y 392.223,Z 540.31,A -85,B 0,C 180,E1 -11712.68,E2 -11712.68} C_VEL
LIN {X 0,Y 392.713,Z 529.664,A -85,B 0,C 180,E1 -11713.849,E2 -11713.849} C_VEL
LIN {X 0,Y 393.233,Z 517.707,A -85,B 0,C 180,E1 -11714.903,E2 -11714.903} C_VEL
LIN {X 0,Y 393.54,Z 505.617,A -85,B 0,C 180,E1 -11715.737,E2 -11715.737} C_VEL
LIN {X 0,Y 393.849,Z 491.535,A -85,B 0,C 180,E1 -11716.456,E2 -11716.456} C_VEL
LIN {X 0,Y 394.031,Z 478.058,A -85,B 0,C 180,E1 -11716.915,E2 -11716.915} C_VEL
LIN {X 0,Y 394.961,Z 415.095,A -85,B 0,C 180,E1 -11718.35,E2 -11718.35} C_VEL
LIN {X 0,Y 390.316,Z 400.81,A -85,B 0,C 180,E1 -11718.886,E2 -11718.886} C_VEL
LIN {X 0,Y 390.112,Z 399.965,A -85,B 0,C 180,E1 -11719.092,E2 -11719.092} C_VEL
LIN {X 0,Y 390.042,Z 399.9,A -85,B 0,C 180,E1 -11722.234,E2 -11722.234} C_VEL
LIN {X 0,Y 390.08,Z 399.893,A -85,B 0,C 180,E1 -11725.62,E2 -11725.62} C_VEL
LIN {X 0,Y 390.035,Z 399.888,A -85,B 0,C 180,E1 -11729.112,E2 -11729.112} C_VEL
LIN {X 0,Y 390.045,Z 399.893,A -85,B 0,C 180,E1 -11732.722,E2 -11732.722} C_VEL
LIN {X 0,Y 390.058,Z 399.896,A -85,B 0,C 180,E1 -11735.825,E2 -11735.825} C_VEL
LIN {X 0,Y 390.07,Z 399.895,A -85,B 0,C 180,E1 -11739.218,E2 -11739.218} C_VEL
LIN {X 0,Y 390.04,Z 399.894,A -85,B 0,C 180,E1 -11742.374,E2 -11742.374} C_VEL
LIN {X 0,Y 390.045,Z 399.894,A -85,B 0,C 180,E1 -11745.354,E2 -11745.354} C_VEL
LIN {X 0,Y 390.028,Z 399.897,A -85,B 0,C 180,E1 -11748.186,E2 -11748.186} C_VEL
LIN {X 0,Y 390.061,Z 399.881,A -85,B 0,C 180,E1 -11750.904,E2 -11750.904} C_VEL
LIN {X 0,Y 390.087,Z 399.882,A -85,B 0,C 180,E1 -11754.793,E2 -11754.793} C_VEL
LIN {X 0,Y 390.129,Z 400.121,A -85,B 0,C 180,E1 -11756.207,E2 -11756.207} C_VEL
LIN {X 0,Y 394.504,Z 416.76,A -85,B 0,C 180,E1 -11759.155,E2 -11759.155} C_VEL
LIN {X 0,Y 396.828,Z 427.207,A -85,B 0,C 180,E1 -11760.921,E2 -11760.921} C_VEL
LIN {X 0,Y 396.752,Z 432.445,A -85,B 0,C 180,E1 -11761.716,E2 -11761.716} C_VEL
LIN {X 0,Y 395.372,Z 454.926,A -85,B 0,C 180,E1 -11765.035,E2 -11765.035} C_VEL
LIN {X 0,Y 394.16,Z 476.942,A -85,B 0,C 180,E1 -11768.179,E2 -11768.179} C_VEL
LIN {X 0,Y 393.679,Z 487.784,A -85,B 0,C 180,E1 -11769.643,E2 -11769.643} C_VEL
LIN {X 0,Y 397.028,Z 510.998,A -85,B 0,C 180,E1 -11770.28,E2 -11770.28} C_VEL
LIN {X 0,Y 395.841,Z 598.72,A -85,B 0,C 180,E1 -11771.898,E2 -11771.898} C_VEL
LIN {X 0,Y 395.315,Z 611.604,A -85,B 0,C 180,E1 -11772.308,E2 -11772.308} C_VEL
LIN {X 0,Y 394.757,Z 624.018,A -85,B 0,C 180,E1 -11772.917,E2 -11772.917} C_VEL
LIN {X 0,Y 393.942,Z 635.571,A -85,B 0,C 180,E1 -11773.681,E2 -11773.681} C_VEL
LIN {X 0,Y 393.06,Z 647.15,A -85,B 0,C 180,E1 -11774.673,E2 -11774.673} C_VEL
LIN {X 0,Y 392.324,Z 657.007,A -85,B 0,C 180,E1 -11775.741,E2 -11775.741} C_VEL
LIN {X 0,Y 391.385,Z 667.156,A -85,B 0,C 180,E1 -11777.103,E2 -11777.103} C_VEL
LIN {X 0,Y 390.525,Z 676.063,A -85,B 0,C 180,E1 -11778.582,E2 -11778.582} C_VEL
LIN {X 0,Y 389.866,Z 683.527,A -85,B 0,C 180,E1 -11780.139,E2 -11780.139} C_VEL
LIN {X 0,Y 389.699,Z 685.775,A -85,B 0,C 180,E1 -11780.679,E2 -11780.679} C_VEL
LIN {X 0,Y 388.804,Z 688.665,A -85,B 0,C 180,E1 -11781.432,E2 -11781.432} C_VEL
LIN {X 0,Y 385.673,Z 692.864,A -85,B 0,C 180,E1 -11782.676,E2 -11782.676} C_VEL
LIN {X 0,Y 382.591,Z 696.409,A -85,B 0,C 180,E1 -11783.981,E2 -11783.981} C_VEL
LIN {X 0,Y 381.786,Z 698.124,A -85,B 0,C 180,E1 -11784.822,E2 -11784.822} C_VEL
LIN {X 0,Y 381.668,Z 699.811,A -85,B 0,C 180,E1 -11785.776,E2 -11785.776} C_VEL
LIN {X 0,Y 381.562,Z 701.24,A -85,B 0,C 180,E1 -11786.833,E2 -11786.833} C_VEL
LIN {X 0,Y 381.561,Z 702.24,A -85,B 0,C 180,E1 -11787.889,E2 -11787.889} C_VEL
LIN {X 0,Y 381.573,Z 703.094,A -85,B 0,C 180,E1 -11790,E2 -11790} C_VEL
LIN {X 0,Y 381.559,Z 702.901,A -85,B 0,C 180,E1 -11791.056,E2 -11791.056} C_VEL
LIN {X 0,Y 381.561,Z 702.313,A -85,B 0,C 180,E1 -11792.111,E2 -11792.111} C_VEL
LIN {X 0,Y 381.666,Z 699.969,A -85,B 0,C 180,E1 -11794.224,E2 -11794.224} C_VEL
LIN {X 0,Y 381.812,Z 696.742,A -85,B 0,C 180,E1 -11795.963,E2 -11795.963} C_VEL
LIN {X 0,Y 382.143,Z 691.589,A -85,B 0,C 180,E1 -11797.928,E2 -11797.928} C_VEL
LIN {X 0,Y 382.652,Z 686.114,A -85,B 0,C 180,E1 -11799.515,E2 -11799.515} C_VEL
LIN {X 0,Y 383.283,Z 679.254,A -85,B 0,C 180,E1 -11801.101,E2 -11801.101} C_VEL
LIN {X 0,Y 384.124,Z 670.674,A -85,B 0,C 180,E1 -11802.683,E2 -11802.683} C_VEL
LIN {X 0,Y 385.067,Z 661.887,A -85,B 0,C 180,E1 -11803.995,E2 -11803.995} C_VEL
LIN {X 0,Y 385.774,Z 652.379,A -85,B 0,C 180,E1 -11805.165,E2 -11805.165} C_VEL
LIN {X 0,Y 386.693,Z 641.547,A -85,B 0,C 180,E1 -11806.227,E2 -11806.227} C_VEL
LIN {X 0,Y 387.641,Z 629.699,A -85,B 0,C 180,E1 -11807.135,E2 -11807.135} C_VEL
LIN {X 0,Y 388.352,Z 617.358,A -85,B 0,C 180,E1 -11807.85,E2 -11807.85} C_VEL
LIN {X 0,Y 388.961,Z 604.357,A -85,B 0,C 180,E1 -11808.365,E2 -11808.365} C_VEL
LIN {X 0,Y 389.333,Z 590.828,A -85,B 0,C 180,E1 -11808.688,E2 -11808.688} C_VEL
LIN {X 0,Y 390.281,Z 510.973,A -85,B 0,C 180,E1 -11810.175,E2 -11810.175} C_VEL
LIN {X 0,Y 386.958,Z 487.945,A -85,B 0,C 180,E1 -11810.818,E2 -11810.818} C_VEL
LIN {X 0,Y 387.86,Z 468.618,A -85,B 0,C 180,E1 -11813.493,E2 -11813.493} C_VEL
LIN {X 0,Y 389.529,Z 442.323,A -85,B 0,C 180,E1 -11817.371,E2 -11817.371} C_VEL
LIN {X 0,Y 390.211,Z 429.538,A -85,B 0,C 180,E1 -11819.302,E2 -11819.302} C_VEL
LIN {X 0,Y 387.357,Z 416.867,A -85,B 0,C 180,E1 -11821.488,E2 -11821.488} C_VEL
LIN {X 0,Y 383.098,Z 401.206,A -85,B 0,C 180,E1 -11824.293,E2 -11824.293} C_VEL
LIN {X 0,Y 383.019,Z 400.802,A -85,B 0,C 180,E1 -11824.458,E2 -11824.458} C_VEL
LIN {X 0,Y 382.994,Z 400.777,A -85,B 0,C 180,E1 -11827.902,E2 -11827.902} C_VEL
LIN {X 0,Y 382.963,Z 400.774,A -85,B 0,C 180,E1 -11831.351,E2 -11831.351} C_VEL
LIN {X 0,Y 382.991,Z 400.757,A -85,B 0,C 180,E1 -11834.302,E2 -11834.302} C_VEL
LIN {X 0,Y 383.013,Z 400.776,A -85,B 0,C 180,E1 -11837.24,E2 -11837.24} C_VEL
LIN {X 0,Y 382.988,Z 400.779,A -85,B 0,C 180,E1 -11840.419,E2 -11840.419} C_VEL
LIN {X 0,Y 383.017,Z 400.776,A -85,B 0,C 180,E1 -11844.043,E2 -11844.043} C_VEL
LIN {X 0,Y 382.989,Z 400.772,A -85,B 0,C 180,E1 -11847.578,E2 -11847.578} C_VEL
LIN {X 0,Y 382.979,Z 400.772,A -85,B 0,C 180,E1 -11850.299,E2 -11850.299} C_VEL
LIN {X 0,Y 383.006,Z 400.777,A -85,B 0,C 180,E1 -11854.045,E2 -11854.045} C_VEL
LIN {X 0,Y 382.992,Z 400.767,A -85,B 0,C 180,E1 -11857.334,E2 -11857.334} C_VEL
LIN {X 0,Y 383.047,Z 400.765,A -85,B 0,C 180,E1 -11860.715,E2 -11860.715} C_VEL
LIN {X 0,Y 383.024,Z 400.771,A -85,B 0,C 180,E1 -11864.024,E2 -11864.024} C_VEL
LIN {X 0,Y 383.138,Z 400.752,A -85,B 0,C 180,E1 -11867.284,E2 -11867.284} C_VEL
LIN {X 0,Y 383.14,Z 400.755,A -85,B 0,C 180,E1 -11870.498,E2 -11870.498} C_VEL
LIN {X 0,Y 383.237,Z 400.739,A -85,B 0,C 180,E1 -11873.683,E2 -11873.683} C_VEL
LIN {X 0,Y 383.376,Z 400.728,A -85,B 0,C 180,E1 -11877.899,E2 -11877.899} C_VEL
LIN {X 0,Y 383.373,Z 400.71,A -85,B 0,C 180,E1 -11882.101,E2 -11882.101} C_VEL
LIN {X 0,Y 383.242,Z 400.745,A -85,B 0,C 180,E1 -11886.317,E2 -11886.317} C_VEL
LIN {X 0,Y 383.14,Z 400.741,A -85,B 0,C 180,E1 -11889.502,E2 -11889.502} C_VEL
LIN {X 0,Y 383.132,Z 400.761,A -85,B 0,C 180,E1 -11893.538,E2 -11893.538} C_VEL
LIN {X 0,Y 383.025,Z 400.757,A -85,B 0,C 180,E1 -11897.419,E2 -11897.419} C_VEL
LIN {X 0,Y 383.015,Z 400.771,A -85,B 0,C 180,E1 -11900.64,E2 -11900.64} C_VEL
LIN {X 0,Y 383.01,Z 400.761,A -85,B 0,C 180,E1 -11903.809,E2 -11903.809} C_VEL
LIN {X 0,Y 382.969,Z 400.779,A -85,B 0,C 180,E1 -11907.309,E2 -11907.309} C_VEL
LIN {X 0,Y 382.984,Z 400.775,A -85,B 0,C 180,E1 -11910.919,E2 -11910.919} C_VEL
LIN {X 0,Y 383.013,Z 400.763,A -85,B 0,C 180,E1 -11914.669,E2 -11914.669} C_VEL
LIN {X 0,Y 382.992,Z 400.775,A -85,B 0,C 180,E1 -11917.902,E2 -11917.902} C_VEL
LIN {X 0,Y 382.961,Z 400.739,A -85,B 0,C 180,E1 -11921.351,E2 -11921.351} C_VEL
LIN {X 0,Y 382.99,Z 400.774,A -85,B 0,C 180,E1 -11924.302,E2 -11924.302} C_VEL
LIN {X 0,Y 382.983,Z 400.764,A -85,B 0,C 180,E1 -11927.236,E2 -11927.236} C_VEL
LIN {X 0,Y 382.985,Z 400.761,A -85,B 0,C 180,E1 -11930.419,E2 -11930.419} C_VEL
LIN {X 0,Y 383.013,Z 400.778,A -85,B 0,C 180,E1 -11934.043,E2 -11934.043} C_VEL
LIN {X 0,Y 383.066,Z 400.903,A -85,B 0,C 180,E1 -11936.257,E2 -11936.257} C_VEL
LIN {X 0,Y 387.522,Z 420.751,A -85,B 0,C 180,E1 -11940.003,E2 -11940.003} C_VEL
LIN {X 0,Y 388.433,Z 424.909,A -85,B 0,C 180,E1 -11940.757,E2 -11940.757} C_VEL
LIN {X 0,Y 388.076,Z 431.817,A -85,B 0,C 180,E1 -11941.91,E2 -11941.91} C_VEL
LIN {X 0,Y 386.284,Z 454.046,A -85,B 0,C 180,E1 -11945.566,E2 -11945.566} C_VEL
LIN {X 0,Y 385.087,Z 471.272,A -85,B 0,C 180,E1 -11948.371,E2 -11948.371} C_VEL
LIN {X 0,Y 386.236,Z 488.196,A -85,B 0,C 180,E1 -11949.33,E2 -11949.33} C_VEL
LIN {X 0,Y 389.748,Z 519.846,A -85,B 0,C 180,E1 -11950.14,E2 -11950.14} C_VEL
LIN {X 0,Y 388.616,Z 606.386,A -85,B 0,C 180,E1 -11951.754,E2 -11951.754} C_VEL
LIN {X 0,Y 387.996,Z 619.637,A -85,B 0,C 180,E1 -11952.201,E2 -11952.201} C_VEL
LIN {X 0,Y 387.388,Z 632.279,A -85,B 0,C 180,E1 -11952.854,E2 -11952.854} C_VEL
LIN {X 0,Y 386.591,Z 643.516,A -85,B 0,C 180,E1 -11953.633,E2 -11953.633} C_VEL
LIN {X 0,Y 385.641,Z 655.067,A -85,B 0,C 180,E1 -11954.677,E2 -11954.677} C_VEL
LIN {X 0,Y 384.81,Z 665.208,A -85,B 0,C 180,E1 -11955.831,E2 -11955.831} C_VEL
LIN {X 0,Y 384.075,Z 673.905,A -85,B 0,C 180,E1 -11957.046,E2 -11957.046} C_VEL
LIN {X 0,Y 383.276,Z 681.681,A -85,B 0,C 180,E1 -11958.363,E2 -11958.363} C_VEL
LIN {X 0,Y 382.675,Z 689.25,A -85,B 0,C 180,E1 -11959.952,E2 -11959.952} C_VEL
LIN {X 0,Y 382.184,Z 695.323,A -85,B 0,C 180,E1 -11961.54,E2 -11961.54} C_VEL
LIN {X 0,Y 381.872,Z 700.116,A -85,B 0,C 180,E1 -11963.129,E2 -11963.129} C_VEL
LIN {X 0,Y 381.784,Z 703.774,A -85,B 0,C 180,E1 -11964.719,E2 -11964.719} C_VEL
LIN {X 0,Y 381.697,Z 705.657,A -85,B 0,C 180,E1 -11965.776,E2 -11965.776} C_VEL
LIN {X 0,Y 381.616,Z 707.078,A -85,B 0,C 180,E1 -11966.833,E2 -11966.833} C_VEL
LIN {X 0,Y 381.637,Z 708.081,A -85,B 0,C 180,E1 -11967.889,E2 -11967.889} C_VEL
LIN {X 0,Y 381.643,Z 708.693,A -85,B 0,C 180,E1 -11968.945,E2 -11968.945} C_VEL
LIN {X 0,Y 381.666,Z 708.912,A -85,B 0,C 180,E1 -11970,E2 -11970} C_VEL
LIN {X 0,Y 381.694,Z 708.69,A -85,B 0,C 180,E1 -11971.055,E2 -11971.055} C_VEL
LIN {X 0,Y 381.623,Z 707.072,A -85,B 0,C 180,E1 -11973.167,E2 -11973.167} C_VEL
LIN {X 0,Y 381.706,Z 705.647,A -85,B 0,C 180,E1 -11974.223,E2 -11974.223} C_VEL
LIN {X 0,Y 381.777,Z 702.434,A -85,B 0,C 180,E1 -11975.917,E2 -11975.917} C_VEL
LIN {X 0,Y 381.965,Z 698.65,A -85,B 0,C 180,E1 -11977.4,E2 -11977.4} C_VEL
LIN {X 0,Y 382.451,Z 692.432,A -85,B 0,C 180,E1 -11979.253,E2 -11979.253} C_VEL
LIN {X 0,Y 382.99,Z 685.643,A -85,B 0,C 180,E1 -11980.841,E2 -11980.841} C_VEL
LIN {X 0,Y 383.576,Z 678.69,A -85,B 0,C 180,E1 -11982.164,E2 -11982.164} C_VEL
LIN {X 0,Y 384.373,Z 670.284,A -85,B 0,C 180,E1 -11983.481,E2 -11983.481} C_VEL
LIN {X 0,Y 385.261,Z 659.87,A -85,B 0,C 180,E1 -11984.797,E2 -11984.797} C_VEL
LIN {X 0,Y 386.084,Z 649.543,A -85,B 0,C 180,E1 -11985.846,E2 -11985.846} C_VEL
LIN {X 0,Y 386.919,Z 638.154,A -85,B 0,C 180,E1 -11986.759,E2 -11986.759} C_VEL
LIN {X 0,Y 387.722,Z 626.326,A -85,B 0,C 180,E1 -11987.471,E2 -11987.471} C_VEL
LIN {X 0,Y 388.317,Z 613.557,A -85,B 0,C 180,E1 -11988.021,E2 -11988.021} C_VEL
LIN {X 0,Y 388.665,Z 599.981,A -85,B 0,C 180,E1 -11988.38,E2 -11988.38} C_VEL
LIN {X 0,Y 388.875,Z 593.247,A -85,B 0,C 180,E1 -11988.54,E2 -11988.54} C_VEL
LIN {X 0,Y 389.607,Z 579.572,A -85,B 0,C 180,E1 -11989.015,E2 -11989.015} C_VEL
LIN {X 0,Y 391.56,Z 519.746,A -85,B 0,C 180,E1 -11990.554,E2 -11990.554} C_VEL
LIN {X 0,Y 389.871,Z 495.292,A -85,B 0,C 180,E1 -11991.423,E2 -11991.423} C_VEL
LIN {X 0,Y 387.476,Z 477.283,A -85,B 0,C 180,E1 -11992.198,E2 -11992.198} C_VEL
LIN {X 0,Y 385.798,Z 467.319,A -85,B 0,C 180,E1 -11992.704,E2 -11992.704} C_VEL
LIN {X 0,Y 387.524,Z 449.758,A -85,B 0,C 180,E1 -11995.802,E2 -11995.802} C_VEL
LIN {X 0,Y 389.939,Z 430.774,A -85,B 0,C 180,E1 -11999.352,E2 -11999.352} C_VEL
LIN {X 0,Y 389.826,Z 427.366,A -85,B 0,C 180,E1 -12000.075,E2 -12000.075} C_VEL
LIN {X 0,Y 387.895,Z 418.128,A -85,B 0,C 180,E1 -12002.309,E2 -12002.309} C_VEL
LIN {X 0,Y 385.502,Z 408.905,A -85,B 0,C 180,E1 -12004.876,E2 -12004.876} C_VEL
LIN {X 0,Y 383.028,Z 400.898,A -85,B 0,C 180,E1 -12007.541,E2 -12007.541} C_VEL
LIN {X 0,Y 382.961,Z 400.783,A -85,B 0,C 180,E1 -12011.199,E2 -12011.199} C_VEL
LIN {X 0,Y 382.989,Z 400.78,A -85,B 0,C 180,E1 -12014.302,E2 -12014.302} C_VEL
LIN {X 0,Y 382.997,Z 400.777,A -85,B 0,C 180,E1 -12017.238,E2 -12017.238} C_VEL
LIN {X 0,Y 382.986,Z 400.777,A -85,B 0,C 180,E1 -12020.419,E2 -12020.419} C_VEL
LIN {X 0,Y 383.024,Z 400.773,A -85,B 0,C 180,E1 -12024.044,E2 -12024.044} C_VEL
LIN {X 0,Y 382.988,Z 400.777,A -85,B 0,C 180,E1 -12027.578,E2 -12027.578} C_VEL
LIN {X 0,Y 382.982,Z 400.78,A -85,B 0,C 180,E1 -12030.299,E2 -12030.299} C_VEL
LIN {X 0,Y 383.015,Z 400.775,A -85,B 0,C 180,E1 -12034.042,E2 -12034.042} C_VEL
LIN {X 0,Y 383.025,Z 400.864,A -85,B 0,C 180,E1 -12037.238,E2 -12037.238} C_VEL
LIN {X 0,Y 383.228,Z 401.846,A -85,B 0,C 180,E1 -12037.488,E2 -12037.488} C_VEL
LIN {X 0,Y 384.708,Z 404.554,A -85,B 0,C 180,E1 -12037.767,E2 -12037.767} C_VEL
LIN {X 0,Y 391.053,Z 416.34,A -85,B 0,C 180,E1 -12038.831,E2 -12038.831} C_VEL
LIN {X 0,Y 394.15,Z 423.242,A -85,B 0,C 180,E1 -12039.353,E2 -12039.353} C_VEL
LIN {X 0,Y 391.87,Z 481.081,A -85,B 0,C 180,E1 -12040.929,E2 -12040.929} C_VEL
LIN {X 0,Y 391.693,Z 495.916,A -85,B 0,C 180,E1 -12041.419,E2 -12041.419} C_VEL
LIN {X 0,Y 391.318,Z 509.643,A -85,B 0,C 180,E1 -12042.113,E2 -12042.113} C_VEL
LIN {X 0,Y 390.764,Z 520.852,A -85,B 0,C 180,E1 -12042.87,E2 -12042.87} C_VEL
LIN {X 0,Y 389.96,Z 532.878,A -85,B 0,C 180,E1 -12043.913,E2 -12043.913} C_VEL
LIN {X 0,Y 389.149,Z 542.5,A -85,B 0,C 180,E1 -12044.953,E2 -12044.953} C_VEL
LIN {X 0,Y 388.347,Z 551.357,A -85,B 0,C 180,E1 -12046.126,E2 -12046.126} C_VEL
LIN {X 0,Y 387.338,Z 560.813,A -85,B 0,C 180,E1 -12047.69,E2 -12047.69} C_VEL
LIN {X 0,Y 386.462,Z 568.245,A -85,B 0,C 180,E1 -12049.231,E2 -12049.231} C_VEL
LIN {X 0,Y 385.673,Z 573.47,A -85,B 0,C 180,E1 -12050.561,E2 -12050.561} C_VEL
LIN {X 0,Y 385.126,Z 578.324,A -85,B 0,C 180,E1 -12052.134,E2 -12052.134} C_VEL
LIN {X 0,Y 384.417,Z 582.03,A -85,B 0,C 180,E1 -12053.702,E2 -12053.702} C_VEL
LIN {X 0,Y 384.123,Z 583.847,A -85,B 0,C 180,E1 -12054.751,E2 -12054.751} C_VEL
LIN {X 0,Y 383.961,Z 585.217,A -85,B 0,C 180,E1 -12055.801,E2 -12055.801} C_VEL
LIN {X 0,Y 383.737,Z 586.177,A -85,B 0,C 180,E1 -12056.85,E2 -12056.85} C_VEL
LIN {X 0,Y 383.55,Z 586.667,A -85,B 0,C 180,E1 -12057.9,E2 -12057.9} C_VEL
LIN {X 0,Y 383.326,Z 586.759,A -85,B 0,C 180,E1 -12058.95,E2 -12058.95} C_VEL
LIN {X 0,Y 383.166,Z 586.44,A -85,B 0,C 180,E1 -12060,E2 -12060} C_VEL
LIN {X 0,Y 383.164,Z 585.643,A -85,B 0,C 180,E1 -12061.051,E2 -12061.051} C_VEL
LIN {X 0,Y 383.093,Z 584.431,A -85,B 0,C 180,E1 -12062.103,E2 -12062.103} C_VEL
LIN {X 0,Y 383.128,Z 581.789,A -85,B 0,C 180,E1 -12063.681,E2 -12063.681} C_VEL
LIN {X 0,Y 383.264,Z 578.098,A -85,B 0,C 180,E1 -12065.261,E2 -12065.261} C_VEL
LIN {X 0,Y 383.567,Z 573.254,A -85,B 0,C 180,E1 -12066.84,E2 -12066.84} C_VEL
LIN {X 0,Y 383.909,Z 567.139,A -85,B 0,C 180,E1 -12068.421,E2 -12068.421} C_VEL
LIN {X 0,Y 384.274,Z 559.481,A -85,B 0,C 180,E1 -12070.006,E2 -12070.006} C_VEL
LIN {X 0,Y 384.824,Z 549.964,A -85,B 0,C 180,E1 -12071.589,E2 -12071.589} C_VEL
LIN {X 0,Y 385.273,Z 540.126,A -85,B 0,C 180,E1 -12072.912,E2 -12072.912} C_VEL
LIN {X 0,Y 385.774,Z 529.211,A -85,B 0,C 180,E1 -12074.103,E2 -12074.103} C_VEL
LIN {X 0,Y 386.267,Z 517.843,A -85,B 0,C 180,E1 -12075.102,E2 -12075.102} C_VEL
LIN {X 0,Y 386.582,Z 505.328,A -85,B 0,C 180,E1 -12075.96,E2 -12075.96} C_VEL
LIN {X 0,Y 386.879,Z 491.627,A -85,B 0,C 180,E1 -12076.659,E2 -12076.659} C_VEL
LIN {X 0,Y 387.088,Z 477.713,A -85,B 0,C 180,E1 -12077.126,E2 -12077.126} C_VEL
LIN {X 0,Y 388.058,Z 416.511,A -85,B 0,C 180,E1 -12078.561,E2 -12078.561} C_VEL
LIN {X 0,Y 383.226,Z 401.631,A -85,B 0,C 180,E1 -12079.128,E2 -12079.128} C_VEL
LIN {X 0,Y 383.096,Z 400.82,A -85,B 0,C 180,E1 -12079.352,E2 -12079.352} C_VEL
LIN {X 0,Y 383.038,Z 400.772,A -85,B 0,C 180,E1 -12083.45,E2 -12083.45} C_VEL
LIN {X 0,Y 383.018,Z 400.773,A -85,B 0,C 180,E1 -12086.128,E2 -12086.128} C_VEL
LIN {X 0,Y 382.982,Z 400.771,A -85,B 0,C 180,E1 -12089.701,E2 -12089.701} C_VEL
LIN {X 0,Y 383.005,Z 400.763,A -85,B 0,C 180,E1 -12093.401,E2 -12093.401} C_VEL
LIN {X 0,Y 383.034,Z 400.772,A -85,B 0,C 180,E1 -12096.165,E2 -12096.165} C_VEL
LIN {X 0,Y 383.009,Z 400.775,A -85,B 0,C 180,E1 -12099.959,E2 -12099.959} C_VEL
LIN {X 0,Y 383.007,Z 400.773,A -85,B 0,C 180,E1 -12102.779,E2 -12102.779} C_VEL
LIN {X 0,Y 382.998,Z 400.773,A -85,B 0,C 180,E1 -12105.789,E2 -12105.789} C_VEL
LIN {X 0,Y 382.987,Z 400.779,A -85,B 0,C 180,E1 -12108.796,E2 -12108.796} C_VEL
LIN {X 0,Y 382.996,Z 400.761,A -85,B 0,C 180,E1 -12112.098,E2 -12112.098} C_VEL
LIN {X 0,Y 383.028,Z 400.761,A -85,B 0,C 180,E1 -12115.333,E2 -12115.333} C_VEL
LIN {X 0,Y 383.104,Z 401.117,A -85,B 0,C 180,E1 -12115.791,E2 -12115.791} C_VEL
LIN {X 0,Y 387.217,Z 416.407,A -85,B 0,C 180,E1 -12118.546,E2 -12118.546} C_VEL
LIN {X 0,Y 390.017,Z 428.817,A -85,B 0,C 180,E1 -12120.695,E2 -12120.695} C_VEL
LIN {X 0,Y 390.021,Z 433.911,A -85,B 0,C 180,E1 -12121.477,E2 -12121.477} C_VEL
LIN {X 0,Y 388.615,Z 455.637,A -85,B 0,C 180,E1 -12124.721,E2 -12124.721} C_VEL
LIN {X 0,Y 387.294,Z 478.932,A -85,B 0,C 180,E1 -12128.07,E2 -12128.07} C_VEL
LIN {X 0,Y 386.897,Z 487.977,A -85,B 0,C 180,E1 -12129.283,E2 -12129.283} C_VEL
LIN {X 0,Y 390.35,Z 511.84,A -85,B 0,C 180,E1 -12129.945,E2 -12129.945} C_VEL
LIN {X 0,Y 389.122,Z 598.711,A -85,B 0,C 180,E1 -12131.575,E2 -12131.575} C_VEL
LIN {X 0,Y 388.571,Z 611.622,A -85,B 0,C 180,E1 -12131.991,E2 -12131.991} C_VEL
LIN {X 0,Y 387.988,Z 624.052,A -85,B 0,C 180,E1 -12132.61,E2 -12132.61} C_VEL
LIN {X 0,Y 387.147,Z 635.612,A -85,B 0,C 180,E1 -12133.387,E2 -12133.387} C_VEL
LIN {X 0,Y 386.189,Z 647.419,A -85,B 0,C 180,E1 -12134.416,E2 -12134.416} C_VEL
LIN {X 0,Y 385.361,Z 658.093,A -85,B 0,C 180,E1 -12135.612,E2 -12135.612} C_VEL
LIN {X 0,Y 384.341,Z 668.458,A -85,B 0,C 180,E1 -12137.056,E2 -12137.056} C_VEL
LIN {X 0,Y 383.425,Z 677.453,A -85,B 0,C 180,E1 -12138.636,E2 -12138.636} C_VEL
LIN {X 0,Y 382.779,Z 684.672,A -85,B 0,C 180,E1 -12140.222,E2 -12140.222} C_VEL
LIN {X 0,Y 382.202,Z 691.298,A -85,B 0,C 180,E1 -12142.073,E2 -12142.073} C_VEL
LIN {X 0,Y 381.848,Z 696.398,A -85,B 0,C 180,E1 -12143.985,E2 -12143.985} C_VEL
LIN {X 0,Y 381.786,Z 698.124,A -85,B 0,C 180,E1 -12144.822,E2 -12144.822} C_VEL
LIN {X 0,Y 380.998,Z 699.669,A -85,B 0,C 180,E1 -12145.675,E2 -12145.675} C_VEL
LIN {X 0,Y 378.018,Z 701.549,A -85,B 0,C 180,E1 -12147.075,E2 -12147.075} C_VEL
LIN {X 0,Y 375.567,Z 702.553,A -85,B 0,C 180,E1 -12148.218,E2 -12148.218} C_VEL
LIN {X 0,Y 374.469,Z 703.04,A -85,B 0,C 180,E1 -12149.26,E2 -12149.26} C_VEL
LIN {X 0,Y 374.449,Z 703.019,A -85,B 0,C 180,E1 -12149.411,E2 -12149.411} C_VEL
LIN {X 0,Y 374.459,Z 702.955,A -85,B 0,C 180,E1 -12151.076,E2 -12151.076} C_VEL
LIN {X 0,Y 374.477,Z 701.394,A -85,B 0,C 180,E1 -12153.228,E2 -12153.228} C_VEL
LIN {X 0,Y 374.598,Z 700.021,A -85,B 0,C 180,E1 -12154.304,E2 -12154.304} C_VEL
LIN {X 0,Y 374.757,Z 696.263,A -85,B 0,C 180,E1 -12156.311,E2 -12156.311} C_VEL
LIN {X 0,Y 375.106,Z 691.64,A -85,B 0,C 180,E1 -12158.078,E2 -12158.078} C_VEL
LIN {X 0,Y 375.635,Z 686.164,A -85,B 0,C 180,E1 -12159.694,E2 -12159.694} C_VEL
LIN {X 0,Y 376.3,Z 679.302,A -85,B 0,C 180,E1 -12161.309,E2 -12161.309} C_VEL
LIN {X 0,Y 377.185,Z 670.72,A -85,B 0,C 180,E1 -12162.92,E2 -12162.92} C_VEL
LIN {X 0,Y 378.166,Z 662.005,A -85,B 0,C 180,E1 -12164.245,E2 -12164.245} C_VEL
LIN {X 0,Y 378.924,Z 652.271,A -85,B 0,C 180,E1 -12165.463,E2 -12165.463} C_VEL
LIN {X 0,Y 379.887,Z 641.58,A -85,B 0,C 180,E1 -12166.526,E2 -12166.526} C_VEL
LIN {X 0,Y 380.86,Z 629.723,A -85,B 0,C 180,E1 -12167.45,E2 -12167.45} C_VEL
LIN {X 0,Y 381.6,Z 617.365,A -85,B 0,C 180,E1 -12168.177,E2 -12168.177} C_VEL
LIN {X 0,Y 382.224,Z 604.335,A -85,B 0,C 180,E1 -12168.701,E2 -12168.701} C_VEL
LIN {X 0,Y 382.633,Z 590.74,A -85,B 0,C 180,E1 -12169.028,E2 -12169.028} C_VEL
LIN {X 0,Y 383.646,Z 511.935,A -85,B 0,C 180,E1 -12170.519,E2 -12170.519} C_VEL
LIN {X 0,Y 380.169,Z 487.655,A -85,B 0,C 180,E1 -12171.23,E2 -12171.23} C_VEL
LIN {X 0,Y 381.258,Z 466.573,A -85,B 0,C 180,E1 -12174.215,E2 -12174.215} C_VEL
LIN {X 0,Y 382.861,Z 442.522,A -85,B 0,C 180,E1 -12177.799,E2 -12177.799} C_VEL
LIN {X 0,Y 383.565,Z 432.384,A -85,B 0,C 180,E1 -12179.35,E2 -12179.35} C_VEL
LIN {X 0,Y 380.985,Z 420.231,A -85,B 0,C 180,E1 -12181.453,E2 -12181.453} C_VEL
LIN {X 0,Y 376.725,Z 404.389,A -85,B 0,C 180,E1 -12184.316,E2 -12184.316} C_VEL
LIN {X 0,Y 376.016,Z 401.836,A -85,B 0,C 180,E1 -12184.832,E2 -12184.832} C_VEL
LIN {X 0,Y 375.937,Z 401.66,A -85,B 0,C 180,E1 -12188.263,E2 -12188.263} C_VEL
LIN {X 0,Y 375.919,Z 401.654,A -85,B 0,C 180,E1 -12191.598,E2 -12191.598} C_VEL
LIN {X 0,Y 375.923,Z 401.635,A -85,B 0,C 180,E1 -12194.73,E2 -12194.73} C_VEL
LIN {X 0,Y 375.928,Z 401.663,A -85,B 0,C 180,E1 -12197.699,E2 -12197.699} C_VEL
LIN {X 0,Y 375.937,Z 401.657,A -85,B 0,C 180,E1 -12200.534,E2 -12200.534} C_VEL
LIN {X 0,Y 375.96,Z 401.648,A -85,B 0,C 180,E1 -12203.497,E2 -12203.497} C_VEL
LIN {X 0,Y 375.96,Z 401.645,A -85,B 0,C 180,E1 -12205.888,E2 -12205.888} C_VEL
LIN {X 0,Y 375.964,Z 401.652,A -85,B 0,C 180,E1 -12209.687,E2 -12209.687} C_VEL
LIN {X 0,Y 375.921,Z 401.654,A -85,B 0,C 180,E1 -12212.135,E2 -12212.135} C_VEL
LIN {X 0,Y 375.972,Z 401.642,A -85,B 0,C 180,E1 -12215.717,E2 -12215.717} C_VEL
LIN {X 0,Y 376.002,Z 401.648,A -85,B 0,C 180,E1 -12219.198,E2 -12219.198} C_VEL
LIN {X 0,Y 376.013,Z 401.632,A -85,B 0,C 180,E1 -12222.599,E2 -12222.599} C_VEL
LIN {X 0,Y 376.093,Z 401.632,A -85,B 0,C 180,E1 -12226.343,E2 -12226.343} C_VEL
LIN {X 0,Y 376.111,Z 401.631,A -85,B 0,C 180,E1 -12230.318,E2 -12230.318} C_VEL
LIN {X 0,Y 376.197,Z 401.618,A -85,B 0,C 180,E1 -12233.564,E2 -12233.564} C_VEL
LIN {X 0,Y 376.34,Z 401.604,A -85,B 0,C 180,E1 -12237.859,E2 -12237.859} C_VEL
LIN {X 0,Y 376.336,Z 401.585,A -85,B 0,C 180,E1 -12242.14,E2 -12242.14} C_VEL
LIN {X 0,Y 376.201,Z 401.622,A -85,B 0,C 180,E1 -12246.436,E2 -12246.436} C_VEL
LIN {X 0,Y 376.11,Z 401.616,A -85,B 0,C 180,E1 -12249.682,E2 -12249.682} C_VEL
LIN {X 0,Y 376.094,Z 401.639,A -85,B 0,C 180,E1 -12253.658,E2 -12253.658} C_VEL
LIN {X 0,Y 375.984,Z 401.635,A -85,B 0,C 180,E1 -12257.576,E2 -12257.576} C_VEL
LIN {X 0,Y 375.982,Z 401.647,A -85,B 0,C 180,E1 -12260.832,E2 -12260.832} C_VEL
LIN {X 0,Y 375.96,Z 401.645,A -85,B 0,C 180,E1 -12264.284,E2 -12264.284} C_VEL
LIN {X 0,Y 375.919,Z 401.65,A -85,B 0,C 180,E1 -12267.865,E2 -12267.865} C_VEL
LIN {X 0,Y 375.959,Z 401.654,A -85,B 0,C 180,E1 -12271.562,E2 -12271.562} C_VEL
LIN {X 0,Y 375.951,Z 401.646,A -85,B 0,C 180,E1 -12275.416,E2 -12275.416} C_VEL
LIN {X 0,Y 375.934,Z 401.65,A -85,B 0,C 180,E1 -12278.262,E2 -12278.262} C_VEL
LIN {X 0,Y 375.914,Z 401.616,A -85,B 0,C 180,E1 -12281.597,E2 -12281.597} C_VEL
LIN {X 0,Y 375.921,Z 401.657,A -85,B 0,C 180,E1 -12284.73,E2 -12284.73} C_VEL
LIN {X 0,Y 375.908,Z 401.635,A -85,B 0,C 180,E1 -12287.696,E2 -12287.696} C_VEL
LIN {X 0,Y 375.934,Z 401.641,A -85,B 0,C 180,E1 -12290.533,E2 -12290.533} C_VEL
LIN {X 0,Y 375.958,Z 401.656,A -85,B 0,C 180,E1 -12293.497,E2 -12293.497} C_VEL
LIN {X 0,Y 376.024,Z 401.855,A -85,B 0,C 180,E1 -12296.025,E2 -12296.025} C_VEL
LIN {X 0,Y 380.831,Z 423.285,A -85,B 0,C 180,E1 -12300.114,E2 -12300.114} C_VEL
LIN {X 0,Y 381.527,Z 426.938,A -85,B 0,C 180,E1 -12300.781,E2 -12300.781} C_VEL
LIN {X 0,Y 380.266,Z 442.302,A -85,B 0,C 180,E1 -12303.372,E2 -12303.372} C_VEL
LIN {X 0,Y 378.676,Z 462.644,A -85,B 0,C 180,E1 -12306.772,E2 -12306.772} C_VEL
LIN {X 0,Y 378.199,Z 469.352,A -85,B 0,C 180,E1 -12307.859,E2 -12307.859} C_VEL
LIN {X 0,Y 379.562,Z 488.818,A -85,B 0,C 180,E1 -12308.969,E2 -12308.969} C_VEL
LIN {X 0,Y 383.086,Z 520.519,A -85,B 0,C 180,E1 -12309.791,E2 -12309.791} C_VEL
LIN {X 0,Y 381.897,Z 606.427,A -85,B 0,C 180,E1 -12311.421,E2 -12311.421} C_VEL
LIN {X 0,Y 381.247,Z 619.633,A -85,B 0,C 180,E1 -12311.876,E2 -12311.876} C_VEL
LIN {X 0,Y 380.606,Z 632.258,A -85,B 0,C 180,E1 -12312.538,E2 -12312.538} C_VEL
LIN {X 0,Y 379.765,Z 643.485,A -85,B 0,C 180,E1 -12313.331,E2 -12313.331} C_VEL
LIN {X 0,Y 378.79,Z 655.029,A -85,B 0,C 180,E1 -12314.393,E2 -12314.393} C_VEL
LIN {X 0,Y 377.879,Z 665.532,A -85,B 0,C 180,E1 -12315.613,E2 -12315.613} C_VEL
LIN {X 0,Y 377.126,Z 673.859,A -85,B 0,C 180,E1 -12316.804,E2 -12316.804} C_VEL
LIN {X 0,Y 376.301,Z 681.633,A -85,B 0,C 180,E1 -12318.144,E2 -12318.144} C_VEL
LIN {X 0,Y 375.647,Z 689.2,A -85,B 0,C 180,E1 -12319.762,E2 -12319.762} C_VEL
LIN {X 0,Y 375.151,Z 695.272,A -85,B 0,C 180,E1 -12321.38,E2 -12321.38} C_VEL
LIN {X 0,Y 374.807,Z 700.064,A -85,B 0,C 180,E1 -12322.999,E2 -12322.999} C_VEL
LIN {X 0,Y 374.68,Z 703.721,A -85,B 0,C 180,E1 -12324.618,E2 -12324.618} C_VEL
LIN {X 0,Y 374.625,Z 705.604,A -85,B 0,C 180,E1 -12325.696,E2 -12325.696} C_VEL
LIN {X 0,Y 374.528,Z 707.025,A -85,B 0,C 180,E1 -12326.773,E2 -12326.773} C_VEL
LIN {X 0,Y 374.535,Z 708.027,A -85,B 0,C 180,E1 -12327.849,E2 -12327.849} C_VEL
LIN {X 0,Y 374.542,Z 708.639,A -85,B 0,C 180,E1 -12328.925,E2 -12328.925} C_VEL
LIN {X 0,Y 374.58,Z 708.858,A -85,B 0,C 180,E1 -12330,E2 -12330} C_VEL
LIN {X 0,Y 374.592,Z 708.636,A -85,B 0,C 180,E1 -12331.075,E2 -12331.075} C_VEL
LIN {X 0,Y 374.535,Z 707.017,A -85,B 0,C 180,E1 -12333.227,E2 -12333.227} C_VEL
LIN {X 0,Y 374.634,Z 705.592,A -85,B 0,C 180,E1 -12334.303,E2 -12334.303} C_VEL
LIN {X 0,Y 374.768,Z 701.694,A -85,B 0,C 180,E1 -12336.327,E2 -12336.327} C_VEL
LIN {X 0,Y 375.026,Z 696.988,A -85,B 0,C 180,E1 -12338.08,E2 -12338.08} C_VEL
LIN {X 0,Y 375.477,Z 691.374,A -85,B 0,C 180,E1 -12339.698,E2 -12339.698} C_VEL
LIN {X 0,Y 376.07,Z 684.298,A -85,B 0,C 180,E1 -12341.316,E2 -12341.316} C_VEL
LIN {X 0,Y 376.95,Z 675.455,A -85,B 0,C 180,E1 -12342.928,E2 -12342.928} C_VEL
LIN {X 0,Y 377.76,Z 666.911,A -85,B 0,C 180,E1 -12344.193,E2 -12344.193} C_VEL
LIN {X 0,Y 378.656,Z 656.217,A -85,B 0,C 180,E1 -12345.474,E2 -12345.474} C_VEL
LIN {X 0,Y 379.592,Z 644.945,A -85,B 0,C 180,E1 -12346.539,E2 -12346.539} C_VEL
LIN {X 0,Y 380.51,Z 633.193,A -85,B 0,C 180,E1 -12347.396,E2 -12347.396} C_VEL
LIN {X 0,Y 381.262,Z 620.162,A -85,B 0,C 180,E1 -12348.089,E2 -12348.089} C_VEL
LIN {X 0,Y 381.797,Z 607.265,A -85,B 0,C 180,E1 -12348.549,E2 -12348.549} C_VEL
LIN {X 0,Y 382.029,Z 596.756,A -85,B 0,C 180,E1 -12348.78,E2 -12348.78} C_VEL
LIN {X 0,Y 383.037,Z 582.528,A -85,B 0,C 180,E1 -12349.355,E2 -12349.355} C_VEL
LIN {X 0,Y 385.23,Z 520.193,A -85,B 0,C 180,E1 -12351.04,E2 -12351.04} C_VEL
LIN {X 0,Y 383.708,Z 496.356,A -85,B 0,C 180,E1 -12351.919,E2 -12351.919} C_VEL
LIN {X 0,Y 381.16,Z 477.296,A -85,B 0,C 180,E1 -12352.781,E2 -12352.781} C_VEL
LIN {X 0,Y 379.203,Z 465.583,A -85,B 0,C 180,E1 -12353.425,E2 -12353.425} C_VEL
LIN {X 0,Y 381.062,Z 448.35,A -85,B 0,C 180,E1 -12356.567,E2 -12356.567} C_VEL
LIN {X 0,Y 383.327,Z 432.232,A -85,B 0,C 180,E1 -12359.671,E2 -12359.671} C_VEL
LIN {X 0,Y 382.898,Z 427.78,A -85,B 0,C 180,E1 -12360.686,E2 -12360.686} C_VEL
LIN {X 0,Y 380.955,Z 418.876,A -85,B 0,C 180,E1 -12362.972,E2 -12362.972} C_VEL
LIN {X 0,Y 378.855,Z 410.979,A -85,B 0,C 180,E1 -12365.291,E2 -12365.291} C_VEL
LIN {X 0,Y 376.817,Z 404.484,A -85,B 0,C 180,E1 -12367.523,E2 -12367.523} C_VEL
LIN {X 0,Y 375.96,Z 401.711,A -85,B 0,C 180,E1 -12368.653,E2 -12368.653} C_VEL
LIN {X 0,Y 375.907,Z 401.66,A -85,B 0,C 180,E1 -12372.304,E2 -12372.304} C_VEL
LIN {X 0,Y 375.92,Z 401.658,A -85,B 0,C 180,E1 -12375.27,E2 -12375.27} C_VEL
LIN {X 0,Y 375.916,Z 401.657,A -85,B 0,C 180,E1 -12378.403,E2 -12378.403} C_VEL
LIN {X 0,Y 375.953,Z 401.653,A -85,B 0,C 180,E1 -12381.91,E2 -12381.91} C_VEL
LIN {X 0,Y 375.981,Z 401.651,A -85,B 0,C 180,E1 -12385.333,E2 -12385.333} C_VEL
LIN {X 0,Y 375.959,Z 401.655,A -85,B 0,C 180,E1 -12388.438,E2 -12388.438} C_VEL
LIN {X 0,Y 375.937,Z 401.658,A -85,B 0,C 180,E1 -12392.137,E2 -12392.137} C_VEL
LIN {X 0,Y 375.985,Z 401.651,A -85,B 0,C 180,E1 -12395.718,E2 -12395.718} C_VEL
LIN {X 0,Y 376.065,Z 401.96,A -85,B 0,C 180,E1 -12396.546,E2 -12396.546} C_VEL
LIN {X 0,Y 376.213,Z 402.707,A -85,B 0,C 180,E1 -12396.685,E2 -12396.685} C_VEL
LIN {X 0,Y 377.75,Z 405.535,A -85,B 0,C 180,E1 -12397.002,E2 -12397.002} C_VEL
LIN {X 0,Y 384.064,Z 416.908,A -85,B 0,C 180,E1 -12398.138,E2 -12398.138} C_VEL
LIN {X 0,Y 388.117,Z 425.255,A -85,B 0,C 180,E1 -12398.844,E2 -12398.844} C_VEL
LIN {X 0,Y 385.644,Z 480.505,A -85,B 0,C 180,E1 -12400.401,E2 -12400.401} C_VEL
LIN {X 0,Y 385.429,Z 496.727,A -85,B 0,C 180,E1 -12400.943,E2 -12400.943} C_VEL
LIN {X 0,Y 385.053,Z 510.432,A -85,B 0,C 180,E1 -12401.642,E2 -12401.642} C_VEL
LIN {X 0,Y 384.444,Z 521.671,A -85,B 0,C 180,E1 -12402.403,E2 -12402.403} C_VEL
LIN {X 0,Y 383.655,Z 532.771,A -85,B 0,C 180,E1 -12403.368,E2 -12403.368} C_VEL
LIN {X 0,Y 382.663,Z 543.639,A -85,B 0,C 180,E1 -12404.555,E2 -12404.555} C_VEL
LIN {X 0,Y 381.725,Z 553.353,A -85,B 0,C 180,E1 -12405.88,E2 -12405.88} C_VEL
LIN {X 0,Y 380.644,Z 562.686,A -85,B 0,C 180,E1 -12407.47,E2 -12407.47} C_VEL
LIN {X 0,Y 379.681,Z 570.144,A -85,B 0,C 180,E1 -12409.077,E2 -12409.077} C_VEL
LIN {X 0,Y 378.857,Z 575.096,A -85,B 0,C 180,E1 -12410.389,E2 -12410.389} C_VEL
LIN {X 0,Y 378.268,Z 579.793,A -85,B 0,C 180,E1 -12411.99,E2 -12411.99} C_VEL
LIN {X 0,Y 377.516,Z 583.401,A -85,B 0,C 180,E1 -12413.587,E2 -12413.587} C_VEL
LIN {X 0,Y 377.179,Z 585.179,A -85,B 0,C 180,E1 -12414.654,E2 -12414.654} C_VEL
LIN {X 0,Y 377.02,Z 586.501,A -85,B 0,C 180,E1 -12415.724,E2 -12415.724} C_VEL
LIN {X 0,Y 376.775,Z 587.385,A -85,B 0,C 180,E1 -12416.792,E2 -12416.792} C_VEL
LIN {X 0,Y 376.571,Z 587.827,A -85,B 0,C 180,E1 -12417.861,E2 -12417.861} C_VEL
LIN {X 0,Y 376.324,Z 587.869,A -85,B 0,C 180,E1 -12418.93,E2 -12418.93} C_VEL
LIN {X 0,Y 376.143,Z 587.477,A -85,B 0,C 180,E1 -12420,E2 -12420} C_VEL
LIN {X 0,Y 376.139,Z 586.606,A -85,B 0,C 180,E1 -12421.071,E2 -12421.071} C_VEL
LIN {X 0,Y 376.07,Z 585.342,A -85,B 0,C 180,E1 -12422.142,E2 -12422.142} C_VEL
LIN {X 0,Y 376.099,Z 582.601,A -85,B 0,C 180,E1 -12423.75,E2 -12423.75} C_VEL
LIN {X 0,Y 376.249,Z 578.806,A -85,B 0,C 180,E1 -12425.359,E2 -12425.359} C_VEL
LIN {X 0,Y 376.553,Z 573.847,A -85,B 0,C 180,E1 -12426.968,E2 -12426.968} C_VEL
LIN {X 0,Y 376.89,Z 567.577,A -85,B 0,C 180,E1 -12428.579,E2 -12428.579} C_VEL
LIN {X 0,Y 377.276,Z 559.743,A -85,B 0,C 180,E1 -12430.193,E2 -12430.193} C_VEL
LIN {X 0,Y 377.838,Z 550.019,A -85,B 0,C 180,E1 -12431.807,E2 -12431.807} C_VEL
LIN {X 0,Y 378.314,Z 539.921,A -85,B 0,C 180,E1 -12433.154,E2 -12433.154} C_VEL
LIN {X 0,Y 378.861,Z 528.741,A -85,B 0,C 180,E1 -12434.366,E2 -12434.366} C_VEL
LIN {X 0,Y 379.301,Z 517.203,A -85,B 0,C 180,E1 -12435.362,E2 -12435.362} C_VEL
LIN {X 0,Y 379.652,Z 503.866,A -85,B 0,C 180,E1 -12436.26,E2 -12436.26} C_VEL
LIN {X 0,Y 379.943,Z 490.623,A -85,B 0,C 180,E1 -12436.903,E2 -12436.903} C_VEL
LIN {X 0,Y 380.108,Z 477.064,A -85,B 0,C 180,E1 -12437.346,E2 -12437.346} C_VEL
LIN {X 0,Y 381.159,Z 417.986,A -85,B 0,C 180,E1 -12438.766,E2 -12438.766} C_VEL
LIN {X 0,Y 376.197,Z 402.545,A -85,B 0,C 180,E1 -12439.361,E2 -12439.361} C_VEL
LIN {X 0,Y 376.039,Z 401.737,A -85,B 0,C 180,E1 -12439.554,E2 -12439.554} C_VEL
LIN {X 0,Y 375.996,Z 401.649,A -85,B 0,C 180,E1 -12443.667,E2 -12443.667} C_VEL
LIN {X 0,Y 375.944,Z 401.655,A -85,B 0,C 180,E1 -12446.658,E2 -12446.658} C_VEL
LIN {X 0,Y 375.964,Z 401.647,A -85,B 0,C 180,E1 -12450.313,E2 -12450.313} C_VEL
LIN {X 0,Y 375.962,Z 401.64,A -85,B 0,C 180,E1 -12454.111,E2 -12454.111} C_VEL
LIN {X 0,Y 375.955,Z 401.654,A -85,B 0,C 180,E1 -12456.741,E2 -12456.741} C_VEL
LIN {X 0,Y 375.989,Z 401.65,A -85,B 0,C 180,E1 -12459.971,E2 -12459.971} C_VEL
LIN {X 0,Y 375.931,Z 401.658,A -85,B 0,C 180,E1 -12463.766,E2 -12463.766} C_VEL
LIN {X 0,Y 375.936,Z 401.658,A -85,B 0,C 180,E1 -12466.811,E2 -12466.811} C_VEL
LIN {X 0,Y 375.945,Z 401.642,A -85,B 0,C 180,E1 -12470.535,E2 -12470.535} C_VEL
LIN {X 0,Y 375.965,Z 401.655,A -85,B 0,C 180,E1 -12473.496,E2 -12473.496} C_VEL
LIN {X 0,Y 376.019,Z 401.872,A -85,B 0,C 180,E1 -12475.29,E2 -12475.29} C_VEL
LIN {X 0,Y 380.028,Z 416.538,A -85,B 0,C 180,E1 -12478.014,E2 -12478.014} C_VEL
LIN {X 0,Y 383.068,Z 429.631,A -85,B 0,C 180,E1 -12480.307,E2 -12480.307} C_VEL
LIN {X 0,Y 383.432,Z 433.501,A -85,B 0,C 180,E1 -12480.94,E2 -12480.94} C_VEL
LIN {X 0,Y 382.049,Z 453.812,A -85,B 0,C 180,E1 -12484.005,E2 -12484.005} C_VEL
LIN {X 0,Y 380.666,Z 476.915,A -85,B 0,C 180,E1 -12487.387,E2 -12487.387} C_VEL
LIN {X 0,Y 380.158,Z 488.037,A -85,B 0,C 180,E1 -12488.902,E2 -12488.902} C_VEL
LIN {X 0,Y 383.649,Z 512.479,A -85,B 0,C 180,E1 -12489.593,E2 -12489.593} C_VEL
LIN {X 0,Y 382.397,Z 598.7,A -85,B 0,C 180,E1 -12491.239,E2 -12491.239} C_VEL
LIN {X 0,Y 381.84,Z 611.641,A -85,B 0,C 180,E1 -12491.662,E2 -12491.662} C_VEL
LIN {X 0,Y 381.229,Z 624.086,A -85,B 0,C 180,E1 -12492.291,E2 -12492.291} C_VEL
LIN {X 0,Y 380.338,Z 635.653,A -85,B 0,C 180,E1 -12493.08,E2 -12493.08} C_VEL
LIN {X 0,Y 379.443,Z 646.369,A -85,B 0,C 180,E1 -12494.021,E2 -12494.021} C_VEL
LIN {X 0,Y 378.552,Z 657.104,A -85,B 0,C 180,E1 -12495.21,E2 -12495.21} C_VEL
LIN {X 0,Y 377.574,Z 666.772,A -85,B 0,C 180,E1 -12496.546,E2 -12496.546} C_VEL
LIN {X 0,Y 376.562,Z 676.168,A -85,B 0,C 180,E1 -12498.153,E2 -12498.153} C_VEL
LIN {X 0,Y 375.857,Z 683.633,A -85,B 0,C 180,E1 -12499.768,E2 -12499.768} C_VEL
LIN {X 0,Y 375.293,Z 689.625,A -85,B 0,C 180,E1 -12501.384,E2 -12501.384} C_VEL
LIN {X 0,Y 374.953,Z 694.367,A -85,B 0,C 180,E1 -12503.002,E2 -12503.002} C_VEL
LIN {X 0,Y 374.701,Z 698.291,A -85,B 0,C 180,E1 -12504.789,E2 -12504.789} C_VEL
LIN {X 0,Y 374.601,Z 699.866,A -85,B 0,C 180,E1 -12505.696,E2 -12505.696} C_VEL
LIN {X 0,Y 374.477,Z 701.294,A -85,B 0,C 180,E1 -12506.773,E2 -12506.773} C_VEL
LIN {X 0,Y 374.459,Z 702.912,A -85,B 0,C 180,E1 -12508.925,E2 -12508.925} C_VEL
LIN {X 0,Y 374.449,Z 703.019,A -85,B 0,C 180,E1 -12509.411,E2 -12509.411} C_VEL
LIN {X 0,Y 373.777,Z 703.132,A -85,B 0,C 180,E1 -12510.309,E2 -12510.309} C_VEL
LIN {X 0,Y 370.885,Z 702.681,A -85,B 0,C 180,E1 -12511.766,E2 -12511.766} C_VEL
LIN {X 0,Y 368.486,Z 701.783,A -85,B 0,C 180,E1 -12512.939,E2 -12512.939} C_VEL
LIN {X 0,Y 367.529,Z 700.794,A -85,B 0,C 180,E1 -12513.841,E2 -12513.841} C_VEL
LIN {X 0,Y 367.49,Z 700.378,A -85,B 0,C 180,E1 -12514.145,E2 -12514.145} C_VEL
LIN {X 0,Y 367.621,Z 698.239,A -85,B 0,C 180,E1 -12515.485,E2 -12515.485} C_VEL
LIN {X 0,Y 367.819,Z 694.674,A -85,B 0,C 180,E1 -12517.135,E2 -12517.135} C_VEL
LIN {X 0,Y 368.236,Z 689.998,A -85,B 0,C 180,E1 -12518.783,E2 -12518.783} C_VEL
LIN {X 0,Y 368.909,Z 682.978,A -85,B 0,C 180,E1 -12520.705,E2 -12520.705} C_VEL
LIN {X 0,Y 369.743,Z 675.29,A -85,B 0,C 180,E1 -12522.348,E2 -12522.348} C_VEL
LIN {X 0,Y 370.835,Z 665.717,A -85,B 0,C 180,E1 -12523.983,E2 -12523.983} C_VEL
LIN {X 0,Y 371.67,Z 657.387,A -85,B 0,C 180,E1 -12525.14,E2 -12525.14} C_VEL
LIN {X 0,Y 372.535,Z 647.263,A -85,B 0,C 180,E1 -12526.297,E2 -12526.297} C_VEL
LIN {X 0,Y 373.638,Z 635.213,A -85,B 0,C 180,E1 -12527.374,E2 -12527.374} C_VEL
LIN {X 0,Y 374.511,Z 623.51,A -85,B 0,C 180,E1 -12528.179,E2 -12528.179} C_VEL
LIN {X 0,Y 375.201,Z 611.539,A -85,B 0,C 180,E1 -12528.781,E2 -12528.781} C_VEL
LIN {X 0,Y 375.713,Z 598.496,A -85,B 0,C 180,E1 -12529.215,E2 -12529.215} C_VEL
LIN {X 0,Y 376.98,Z 512.43,A -85,B 0,C 180,E1 -12530.887,E2 -12530.887} C_VEL
LIN {X 0,Y 373.404,Z 487.644,A -85,B 0,C 180,E1 -12531.634,E2 -12531.634} C_VEL
LIN {X 0,Y 374.459,Z 468.332,A -85,B 0,C 180,E1 -12534.388,E2 -12534.388} C_VEL
LIN {X 0,Y 376.129,Z 444.036,A -85,B 0,C 180,E1 -12538.049,E2 -12538.049} C_VEL
LIN {X 0,Y 376.792,Z 433.818,A -85,B 0,C 180,E1 -12539.623,E2 -12539.623} C_VEL
LIN {X 0,Y 374.205,Z 421.916,A -85,B 0,C 180,E1 -12541.727,E2 -12541.727} C_VEL
LIN {X 0,Y 370.058,Z 406.53,A -85,B 0,C 180,E1 -12544.559,E2 -12544.559} C_VEL
LIN {X 0,Y 368.952,Z 402.672,A -85,B 0,C 180,E1 -12545.346,E2 -12545.346} C_VEL
LIN {X 0,Y 368.876,Z 402.533,A -85,B 0,C 180,E1 -12548.957,E2 -12548.957} C_VEL
LIN {X 0,Y 368.873,Z 402.538,A -85,B 0,C 180,E1 -12552.008,E2 -12552.008} C_VEL
LIN {X 0,Y 368.878,Z 402.513,A -85,B 0,C 180,E1 -12555.175,E2 -12555.175} C_VEL
LIN {X 0,Y 368.872,Z 402.537,A -85,B 0,C 180,E1 -12558.176,E2 -12558.176} C_VEL
LIN {X 0,Y 368.879,Z 402.538,A -85,B 0,C 180,E1 -12561.366,E2 -12561.366} C_VEL
LIN {X 0,Y 368.933,Z 402.529,A -85,B 0,C 180,E1 -12565.146,E2 -12565.146} C_VEL
LIN {X 0,Y 368.916,Z 402.532,A -85,B 0,C 180,E1 -12569.045,E2 -12569.045} C_VEL
LIN {X 0,Y 368.91,Z 402.522,A -85,B 0,C 180,E1 -12571.558,E2 -12571.558} C_VEL
LIN {X 0,Y 368.926,Z 402.526,A -85,B 0,C 180,E1 -12575.222,E2 -12575.222} C_VEL
LIN {X 0,Y 368.923,Z 402.529,A -85,B 0,C 180,E1 -12578.981,E2 -12578.981} C_VEL
LIN {X 0,Y 368.956,Z 402.509,A -85,B 0,C 180,E1 -12582.255,E2 -12582.255} C_VEL
LIN {X 0,Y 369.041,Z 402.512,A -85,B 0,C 180,E1 -12586.228,E2 -12586.228} C_VEL
LIN {X 0,Y 369.061,Z 402.505,A -85,B 0,C 180,E1 -12590.131,E2 -12590.131} C_VEL
LIN {X 0,Y 369.159,Z 402.496,A -85,B 0,C 180,E1 -12593.441,E2 -12593.441} C_VEL
LIN {X 0,Y 369.304,Z 402.479,A -85,B 0,C 180,E1 -12597.819,E2 -12597.819} C_VEL
LIN {X 0,Y 369.299,Z 402.461,A -85,B 0,C 180,E1 -12602.181,E2 -12602.181} C_VEL
LIN {X 0,Y 369.162,Z 402.498,A -85,B 0,C 180,E1 -12606.559,E2 -12606.559} C_VEL
LIN {X 0,Y 369.061,Z 402.493,A -85,B 0,C 180,E1 -12609.868,E2 -12609.868} C_VEL
LIN {X 0,Y 369.041,Z 402.516,A -85,B 0,C 180,E1 -12613.772,E2 -12613.772} C_VEL
LIN {X 0,Y 368.939,Z 402.514,A -85,B 0,C 180,E1 -12617.745,E2 -12617.745} C_VEL
LIN {X 0,Y 368.911,Z 402.529,A -85,B 0,C 180,E1 -12621.221,E2 -12621.221} C_VEL
LIN {X 0,Y 368.919,Z 402.516,A -85,B 0,C 180,E1 -12623.876,E2 -12623.876} C_VEL
LIN {X 0,Y 368.859,Z 402.537,A -85,B 0,C 180,E1 -12627.212,E2 -12627.212} C_VEL
LIN {X 0,Y 368.895,Z 402.52,A -85,B 0,C 180,E1 -12629.692,E2 -12629.692} C_VEL
LIN {X 0,Y 368.899,Z 402.53,A -85,B 0,C 180,E1 -12633.043,E2 -12633.043} C_VEL
LIN {X 0,Y 368.913,Z 402.533,A -85,B 0,C 180,E1 -12636.197,E2 -12636.197} C_VEL
LIN {X 0,Y 368.874,Z 402.524,A -85,B 0,C 180,E1 -12638.957,E2 -12638.957} C_VEL
LIN {X 0,Y 368.859,Z 402.495,A -85,B 0,C 180,E1 -12642.005,E2 -12642.005} C_VEL
LIN {X 0,Y 368.874,Z 402.535,A -85,B 0,C 180,E1 -12645.174,E2 -12645.174} C_VEL
LIN {X 0,Y 368.861,Z 402.505,A -85,B 0,C 180,E1 -12648.174,E2 -12648.174} C_VEL
LIN {X 0,Y 368.876,Z 402.533,A -85,B 0,C 180,E1 -12651.366,E2 -12651.366} C_VEL
LIN {X 0,Y 368.931,Z 402.531,A -85,B 0,C 180,E1 -12655.146,E2 -12655.146} C_VEL
LIN {X 0,Y 368.974,Z 402.763,A -85,B 0,C 180,E1 -12655.771,E2 -12655.771} C_VEL
LIN {X 0,Y 373.714,Z 423.956,A -85,B 0,C 180,E1 -12659.891,E2 -12659.891} C_VEL
LIN {X 0,Y 374.556,Z 428.88,A -85,B 0,C 180,E1 -12660.8,E2 -12660.8} C_VEL
LIN {X 0,Y 372.993,Z 445.901,A -85,B 0,C 180,E1 -12663.718,E2 -12663.718} C_VEL
LIN {X 0,Y 371.475,Z 464.653,A -85,B 0,C 180,E1 -12666.914,E2 -12666.914} C_VEL
LIN {X 0,Y 371.319,Z 467.488,A -85,B 0,C 180,E1 -12667.327,E2 -12667.327} C_VEL
LIN {X 0,Y 372.906,Z 489.209,A -85,B 0,C 180,E1 -12668.581,E2 -12668.581} C_VEL
LIN {X 0,Y 376.343,Z 519.942,A -85,B 0,C 180,E1 -12669.4,E2 -12669.4} C_VEL
LIN {X 0,Y 375.346,Z 595.278,A -85,B 0,C 180,E1 -12670.837,E2 -12670.837} C_VEL
LIN {X 0,Y 374.964,Z 610.931,A -85,B 0,C 180,E1 -12671.207,E2 -12671.207} C_VEL
LIN {X 0,Y 374.341,Z 622.603,A -85,B 0,C 180,E1 -12671.671,E2 -12671.671} C_VEL
LIN {X 0,Y 373.685,Z 634.31,A -85,B 0,C 180,E1 -12672.346,E2 -12672.346} C_VEL
LIN {X 0,Y 372.705,Z 646.59,A -85,B 0,C 180,E1 -12673.287,E2 -12673.287} C_VEL
LIN {X 0,Y 371.753,Z 657.534,A -85,B 0,C 180,E1 -12674.371,E2 -12674.371} C_VEL
LIN {X 0,Y 370.729,Z 668.332,A -85,B 0,C 180,E1 -12675.733,E2 -12675.733} C_VEL
LIN {X 0,Y 369.876,Z 677.085,A -85,B 0,C 180,E1 -12677.099,E2 -12677.099} C_VEL
LIN {X 0,Y 369.059,Z 684.287,A -85,B 0,C 180,E1 -12678.466,E2 -12678.466} C_VEL
LIN {X 0,Y 368.458,Z 691.352,A -85,B 0,C 180,E1 -12680.115,E2 -12680.115} C_VEL
LIN {X 0,Y 367.953,Z 696.962,A -85,B 0,C 180,E1 -12681.764,E2 -12681.764} C_VEL
LIN {X 0,Y 367.607,Z 702.224,A -85,B 0,C 180,E1 -12683.8,E2 -12683.8} C_VEL
LIN {X 0,Y 367.554,Z 705.551,A -85,B 0,C 180,E1 -12685.613,E2 -12685.613} C_VEL
LIN {X 0,Y 367.444,Z 706.971,A -85,B 0,C 180,E1 -12686.71,E2 -12686.71} C_VEL
LIN {X 0,Y 367.433,Z 707.973,A -85,B 0,C 180,E1 -12687.807,E2 -12687.807} C_VEL
LIN {X 0,Y 367.441,Z 708.585,A -85,B 0,C 180,E1 -12688.904,E2 -12688.904} C_VEL
LIN {X 0,Y 367.48,Z 708.804,A -85,B 0,C 180,E1 -12690,E2 -12690} C_VEL
LIN {X 0,Y 367.49,Z 708.582,A -85,B 0,C 180,E1 -12691.096,E2 -12691.096} C_VEL
LIN {X 0,Y 367.451,Z 706.963,A -85,B 0,C 180,E1 -12693.289,E2 -12693.289} C_VEL
LIN {X 0,Y 367.563,Z 705.538,A -85,B 0,C 180,E1 -12694.386,E2 -12694.386} C_VEL
LIN {X 0,Y 367.691,Z 701.934,A -85,B 0,C 180,E1 -12696.319,E2 -12696.319} C_VEL
LIN {X 0,Y 367.967,Z 696.935,A -85,B 0,C 180,E1 -12698.236,E2 -12698.236} C_VEL
LIN {X 0,Y 368.464,Z 691.321,A -85,B 0,C 180,E1 -12699.885,E2 -12699.885} C_VEL
LIN {X 0,Y 369.071,Z 684.246,A -85,B 0,C 180,E1 -12701.534,E2 -12701.534} C_VEL
LIN {X 0,Y 370.011,Z 675.404,A -85,B 0,C 180,E1 -12703.175,E2 -12703.175} C_VEL
LIN {X 0,Y 370.978,Z 665.783,A -85,B 0,C 180,E1 -12704.609,E2 -12704.609} C_VEL
LIN {X 0,Y 371.941,Z 654.892,A -85,B 0,C 180,E1 -12705.901,E2 -12705.901} C_VEL
LIN {X 0,Y 372.925,Z 643.328,A -85,B 0,C 180,E1 -12706.984,E2 -12706.984} C_VEL
LIN {X 0,Y 373.878,Z 630.947,A -85,B 0,C 180,E1 -12707.857,E2 -12707.857} C_VEL
LIN {X 0,Y 374.604,Z 617.899,A -85,B 0,C 180,E1 -12708.528,E2 -12708.528} C_VEL
LIN {X 0,Y 375.162,Z 604.605,A -85,B 0,C 180,E1 -12708.96,E2 -12708.96} C_VEL
LIN {X 0,Y 375.326,Z 598.15,A -85,B 0,C 180,E1 -12709.128,E2 -12709.128} C_VEL
LIN {X 0,Y 376.541,Z 583.544,A -85,B 0,C 180,E1 -12709.773,E2 -12709.773} C_VEL
LIN {X 0,Y 377.563,Z 558.458,A -85,B 0,C 180,E1 -12710.498,E2 -12710.498} C_VEL
LIN {X 0,Y 379.016,Z 521.172,A -85,B 0,C 180,E1 -12711.533,E2 -12711.533} C_VEL
LIN {X 0,Y 377.636,Z 497.677,A -85,B 0,C 180,E1 -12712.433,E2 -12712.433} C_VEL
LIN {X 0,Y 375.295,Z 479.345,A -85,B 0,C 180,E1 -12713.299,E2 -12713.299} C_VEL
LIN {X 0,Y 372.722,Z 463.903,A -85,B 0,C 180,E1 -12714.175,E2 -12714.175} C_VEL
LIN {X 0,Y 374.952,Z 445.579,A -85,B 0,C 180,E1 -12717.64,E2 -12717.64} C_VEL
LIN {X 0,Y 376.701,Z 434.071,A -85,B 0,C 180,E1 -12719.938,E2 -12719.938} C_VEL
LIN {X 0,Y 376.345,Z 430.425,A -85,B 0,C 180,E1 -12720.793,E2 -12720.793} C_VEL
LIN {X 0,Y 374.62,Z 422.174,A -85,B 0,C 180,E1 -12722.96,E2 -12722.96} C_VEL
LIN {X 0,Y 372.562,Z 414.219,A -85,B 0,C 180,E1 -12725.36,E2 -12725.36} C_VEL
LIN {X 0,Y 370.487,Z 407.561,A -85,B 0,C 180,E1 -12727.713,E2 -12727.713} C_VEL
LIN {X 0,Y 368.918,Z 402.594,A -85,B 0,C 180,E1 -12729.834,E2 -12729.834} C_VEL
LIN {X 0,Y 368.878,Z 402.535,A -85,B 0,C 180,E1 -12733.615,E2 -12733.615} C_VEL
LIN {X 0,Y 368.883,Z 402.533,A -85,B 0,C 180,E1 -12736.695,E2 -12736.695} C_VEL
LIN {X 0,Y 368.884,Z 402.535,A -85,B 0,C 180,E1 -12739.648,E2 -12739.648} C_VEL
LIN {X 0,Y 368.9,Z 402.535,A -85,B 0,C 180,E1 -12743.145,E2 -12743.145} C_VEL
LIN {X 0,Y 368.898,Z 402.535,A -85,B 0,C 180,E1 -12746.462,E2 -12746.462} C_VEL
LIN {X 0,Y 368.931,Z 402.528,A -85,B 0,C 180,E1 -12749.047,E2 -12749.047} C_VEL
LIN {X 0,Y 368.877,Z 402.535,A -85,B 0,C 180,E1 -12752.79,E2 -12752.79} C_VEL
LIN {X 0,Y 368.976,Z 402.752,A -85,B 0,C 180,E1 -12755.605,E2 -12755.605} C_VEL
LIN {X 0,Y 369.266,Z 403.913,A -85,B 0,C 180,E1 -12755.835,E2 -12755.835} C_VEL
LIN {X 0,Y 370.751,Z 406.438,A -85,B 0,C 180,E1 -12756.147,E2 -12756.147} C_VEL
LIN {X 0,Y 371.604,Z 407.695,A -85,B 0,C 180,E1 -12756.314,E2 -12756.314} C_VEL
LIN {X 0,Y 377.86,Z 418.873,A -85,B 0,C 180,E1 -12757.524,E2 -12757.524} C_VEL
LIN {X 0,Y 382.141,Z 427.575,A -85,B 0,C 180,E1 -12758.311,E2 -12758.311} C_VEL
LIN {X 0,Y 379.55,Z 480.757,A -85,B 0,C 180,E1 -12759.861,E2 -12759.861} C_VEL
LIN {X 0,Y 379.25,Z 497.79,A -85,B 0,C 180,E1 -12760.444,E2 -12760.444} C_VEL
LIN {X 0,Y 378.842,Z 511.32,A -85,B 0,C 180,E1 -12761.152,E2 -12761.152} C_VEL
LIN {X 0,Y 378.105,Z 523.551,A -85,B 0,C 180,E1 -12762.003,E2 -12762.003} C_VEL
LIN {X 0,Y 377.198,Z 535.404,A -85,B 0,C 180,E1 -12763.075,E2 -12763.075} C_VEL
LIN {X 0,Y 376.238,Z 544.965,A -85,B 0,C 180,E1 -12764.146,E2 -12764.146} C_VEL
LIN {X 0,Y 375.33,Z 553.762,A -85,B 0,C 180,E1 -12765.358,E2 -12765.358} C_VEL
LIN {X 0,Y 374.361,Z 561.775,A -85,B 0,C 180,E1 -12766.705,E2 -12766.705} C_VEL
LIN {X 0,Y 373.287,Z 569.237,A -85,B 0,C 180,E1 -12768.244,E2 -12768.244} C_VEL
LIN {X 0,Y 372.443,Z 574.855,A -85,B 0,C 180,E1 -12769.673,E2 -12769.673} C_VEL
LIN {X 0,Y 371.562,Z 579.933,A -85,B 0,C 180,E1 -12771.297,E2 -12771.297} C_VEL
LIN {X 0,Y 370.93,Z 583.768,A -85,B 0,C 180,E1 -12772.926,E2 -12772.926} C_VEL
LIN {X 0,Y 370.26,Z 586.534,A -85,B 0,C 180,E1 -12774.554,E2 -12774.554} C_VEL
LIN {X 0,Y 370.073,Z 587.786,A -85,B 0,C 180,E1 -12775.643,E2 -12775.643} C_VEL
LIN {X 0,Y 369.808,Z 588.586,A -85,B 0,C 180,E1 -12776.732,E2 -12776.732} C_VEL
LIN {X 0,Y 369.588,Z 588.978,A -85,B 0,C 180,E1 -12777.82,E2 -12777.82} C_VEL
LIN {X 0,Y 369.32,Z 588.972,A -85,B 0,C 180,E1 -12778.91,E2 -12778.91} C_VEL
LIN {X 0,Y 369.117,Z 588.495,A -85,B 0,C 180,E1 -12780,E2 -12780} C_VEL
LIN {X 0,Y 369.113,Z 587.566,A -85,B 0,C 180,E1 -12781.091,E2 -12781.091} C_VEL
LIN {X 0,Y 369.046,Z 586.239,A -85,B 0,C 180,E1 -12782.183,E2 -12782.183} C_VEL
LIN {X 0,Y 369.07,Z 583.387,A -85,B 0,C 180,E1 -12783.822,E2 -12783.822} C_VEL
LIN {X 0,Y 369.235,Z 579.469,A -85,B 0,C 180,E1 -12785.461,E2 -12785.461} C_VEL
LIN {X 0,Y 369.575,Z 573.462,A -85,B 0,C 180,E1 -12787.352,E2 -12787.352} C_VEL
LIN {X 0,Y 369.933,Z 567.148,A -85,B 0,C 180,E1 -12788.922,E2 -12788.922} C_VEL
LIN {X 0,Y 370.281,Z 559.957,A -85,B 0,C 180,E1 -12790.388,E2 -12790.388} C_VEL
LIN {X 0,Y 370.79,Z 551.834,A -85,B 0,C 180,E1 -12791.757,E2 -12791.757} C_VEL
LIN {X 0,Y 371.22,Z 541.928,A -85,B 0,C 180,E1 -12793.132,E2 -12793.132} C_VEL
LIN {X 0,Y 371.764,Z 530.949,A -85,B 0,C 180,E1 -12794.366,E2 -12794.366} C_VEL
LIN {X 0,Y 372.317,Z 519.115,A -85,B 0,C 180,E1 -12795.432,E2 -12795.432} C_VEL
LIN {X 0,Y 372.631,Z 506.634,A -85,B 0,C 180,E1 -12796.309,E2 -12796.309} C_VEL
LIN {X 0,Y 372.973,Z 493.047,A -85,B 0,C 180,E1 -12797.017,E2 -12797.017} C_VEL
LIN {X 0,Y 373.168,Z 479.002,A -85,B 0,C 180,E1 -12797.502,E2 -12797.502} C_VEL
LIN {X 0,Y 374.169,Z 419.154,A -85,B 0,C 180,E1 -12798.985,E2 -12798.985} C_VEL
LIN {X 0,Y 369.146,Z 403.371,A -85,B 0,C 180,E1 -12799.614,E2 -12799.614} C_VEL
LIN {X 0,Y 368.973,Z 402.613,A -85,B 0,C 180,E1 -12799.809,E2 -12799.809} C_VEL
LIN {X 0,Y 368.943,Z 402.527,A -85,B 0,C 180,E1 -12803.886,E2 -12803.886} C_VEL
LIN {X 0,Y 368.881,Z 402.529,A -85,B 0,C 180,E1 -12807.21,E2 -12807.21} C_VEL
LIN {X 0,Y 368.931,Z 402.531,A -85,B 0,C 180,E1 -12810.954,E2 -12810.954} C_VEL
LIN {X 0,Y 368.931,Z 402.524,A -85,B 0,C 180,E1 -12815.001,E2 -12815.001} C_VEL
LIN {X 0,Y 368.909,Z 402.524,A -85,B 0,C 180,E1 -12818.64,E2 -12818.64} C_VEL
LIN {X 0,Y 368.881,Z 402.528,A -85,B 0,C 180,E1 -12822.009,E2 -12822.009} C_VEL
LIN {X 0,Y 368.881,Z 402.529,A -85,B 0,C 180,E1 -12825.176,E2 -12825.176} C_VEL
LIN {X 0,Y 368.882,Z 402.531,A -85,B 0,C 180,E1 -12828.177,E2 -12828.177} C_VEL
LIN {X 0,Y 368.88,Z 402.516,A -85,B 0,C 180,E1 -12831.366,E2 -12831.366} C_VEL
LIN {X 0,Y 368.941,Z 402.688,A -85,B 0,C 180,E1 -12834.774,E2 -12834.774} C_VEL
LIN {X 0,Y 372.144,Z 414.016,A -85,B 0,C 180,E1 -12836.95,E2 -12836.95} C_VEL
LIN {X 0,Y 375.808,Z 429.084,A -85,B 0,C 180,E1 -12839.673,E2 -12839.673} C_VEL
LIN {X 0,Y 376.618,Z 433.048,A -85,B 0,C 180,E1 -12840.362,E2 -12840.362} C_VEL
LIN {X 0,Y 376.427,Z 439.334,A -85,B 0,C 180,E1 -12841.343,E2 -12841.343} C_VEL
LIN {X 0,Y 374.84,Z 461.796,A -85,B 0,C 180,E1 -12844.751,E2 -12844.751} C_VEL
LIN {X 0,Y 373.479,Z 484.444,A -85,B 0,C 180,E1 -12848.038,E2 -12848.038} C_VEL
LIN {X 0,Y 373.342,Z 487.826,A -85,B 0,C 180,E1 -12848.486,E2 -12848.486} C_VEL
LIN {X 0,Y 377.034,Z 513.448,A -85,B 0,C 180,E1 -12849.239,E2 -12849.239} C_VEL
LIN {X 0,Y 375.688,Z 598.689,A -85,B 0,C 180,E1 -12850.891,E2 -12850.891} C_VEL
LIN {X 0,Y 375.119,Z 611.66,A -85,B 0,C 180,E1 -12851.321,E2 -12851.321} C_VEL
LIN {X 0,Y 374.483,Z 624.12,A -85,B 0,C 180,E1 -12851.961,E2 -12851.961} C_VEL
LIN {X 0,Y 373.55,Z 635.694,A -85,B 0,C 180,E1 -12852.763,E2 -12852.763} C_VEL
LIN {X 0,Y 372.599,Z 646.414,A -85,B 0,C 180,E1 -12853.72,E2 -12853.72} C_VEL
LIN {X 0,Y 371.656,Z 657.173,A -85,B 0,C 180,E1 -12854.932,E2 -12854.932} C_VEL
LIN {X 0,Y 370.671,Z 666.823,A -85,B 0,C 180,E1 -12856.29,E2 -12856.29} C_VEL
LIN {X 0,Y 369.596,Z 676.22,A -85,B 0,C 180,E1 -12857.926,E2 -12857.926} C_VEL
LIN {X 0,Y 368.87,Z 683.686,A -85,B 0,C 180,E1 -12859.572,E2 -12859.572} C_VEL
LIN {X 0,Y 368.252,Z 689.679,A -85,B 0,C 180,E1 -12861.218,E2 -12861.218} C_VEL
LIN {X 0,Y 367.893,Z 694.421,A -85,B 0,C 180,E1 -12862.867,E2 -12862.867} C_VEL
LIN {X 0,Y 367.637,Z 698.051,A -85,B 0,C 180,E1 -12864.515,E2 -12864.515} C_VEL
LIN {X 0,Y 367.536,Z 699.92,A -85,B 0,C 180,E1 -12865.613,E2 -12865.613} C_VEL
LIN {X 0,Y 367.397,Z 701.349,A -85,B 0,C 180,E1 -12866.71,E2 -12866.71} C_VEL
LIN {X 0,Y 367.359,Z 702.966,A -85,B 0,C 180,E1 -12868.904,E2 -12868.904} C_VEL
LIN {X 0,Y 367.374,Z 703.202,A -85,B 0,C 180,E1 -12870,E2 -12870} C_VEL
LIN {X 0,Y 367.359,Z 703.009,A -85,B 0,C 180,E1 -12871.096,E2 -12871.096} C_VEL
LIN {X 0,Y 367.396,Z 701.447,A -85,B 0,C 180,E1 -12873.29,E2 -12873.29} C_VEL
LIN {X 0,Y 367.49,Z 700.378,A -85,B 0,C 180,E1 -12874.145,E2 -12874.145} C_VEL
LIN {X 0,Y 366.939,Z 699.109,A -85,B 0,C 180,E1 -12875.04,E2 -12875.04} C_VEL
LIN {X 0,Y 364.21,Z 696.467,A -85,B 0,C 180,E1 -12876.478,E2 -12876.478} C_VEL
LIN {X 0,Y 361.951,Z 693.827,A -85,B 0,C 180,E1 -12877.613,E2 -12877.613} C_VEL
LIN {X 0,Y 361.123,Z 691.528,A -85,B 0,C 180,E1 -12878.47,E2 -12878.47} C_VEL
LIN {X 0,Y 361.136,Z 690.658,A -85,B 0,C 180,E1 -12878.754,E2 -12878.754} C_VEL
LIN {X 0,Y 361.803,Z 684.123,A -85,B 0,C 180,E1 -12880.634,E2 -12880.634} C_VEL
LIN {X 0,Y 362.588,Z 676.753,A -85,B 0,C 180,E1 -12882.311,E2 -12882.311} C_VEL
LIN {X 0,Y 363.55,Z 669.219,A -85,B 0,C 180,E1 -12883.699,E2 -12883.699} C_VEL
LIN {X 0,Y 364.661,Z 659.392,A -85,B 0,C 180,E1 -12885.168,E2 -12885.168} C_VEL
LIN {X 0,Y 365.435,Z 649.851,A -85,B 0,C 180,E1 -12886.336,E2 -12886.336} C_VEL
LIN {X 0,Y 366.564,Z 638.598,A -85,B 0,C 180,E1 -12887.432,E2 -12887.432} C_VEL
LIN {X 0,Y 367.54,Z 626.741,A -85,B 0,C 180,E1 -12888.32,E2 -12888.32} C_VEL
LIN {X 0,Y 368.348,Z 613.838,A -85,B 0,C 180,E1 -12889.035,E2 -12889.035} C_VEL
LIN {X 0,Y 368.953,Z 601.053,A -85,B 0,C 180,E1 -12889.509,E2 -12889.509} C_VEL
LIN {X 0,Y 369.743,Z 559.244,A -85,B 0,C 180,E1 -12890.356,E2 -12890.356} C_VEL
LIN {X 0,Y 370.353,Z 513.337,A -85,B 0,C 180,E1 -12891.258,E2 -12891.258} C_VEL
LIN {X 0,Y 366.682,Z 487.975,A -85,B 0,C 180,E1 -12892.021,E2 -12892.021} C_VEL
LIN {X 0,Y 367.231,Z 477.273,A -85,B 0,C 180,E1 -12893.524,E2 -12893.524} C_VEL
LIN {X 0,Y 368.852,Z 452.666,A -85,B 0,C 180,E1 -12897.213,E2 -12897.213} C_VEL
LIN {X 0,Y 370.038,Z 437.291,A -85,B 0,C 180,E1 -12899.592,E2 -12899.592} C_VEL
LIN {X 0,Y 369.623,Z 433.324,A -85,B 0,C 180,E1 -12900.257,E2 -12900.257} C_VEL
LIN {X 0,Y 366.83,Z 421.286,A -85,B 0,C 180,E1 -12902.442,E2 -12902.442} C_VEL
LIN {X 0,Y 363.521,Z 409.057,A -85,B 0,C 180,E1 -12904.748,E2 -12904.748} C_VEL
LIN {X 0,Y 361.902,Z 403.586,A -85,B 0,C 180,E1 -12905.847,E2 -12905.847} C_VEL
LIN {X 0,Y 361.828,Z 403.409,A -85,B 0,C 180,E1 -12909.018,E2 -12909.018} C_VEL
LIN {X 0,Y 361.834,Z 403.414,A -85,B 0,C 180,E1 -12912.83,E2 -12912.83} C_VEL
LIN {X 0,Y 361.818,Z 403.4,A -85,B 0,C 180,E1 -12915.947,E2 -12915.947} C_VEL
LIN {X 0,Y 361.815,Z 403.412,A -85,B 0,C 180,E1 -12919.249,E2 -12919.249} C_VEL
LIN {X 0,Y 361.864,Z 403.4,A -85,B 0,C 180,E1 -12922.981,E2 -12922.981} C_VEL
LIN {X 0,Y 361.861,Z 403.397,A -85,B 0,C 180,E1 -12926.631,E2 -12926.631} C_VEL
LIN {X 0,Y 361.858,Z 403.409,A -85,B 0,C 180,E1 -12929.67,E2 -12929.67} C_VEL
LIN {X 0,Y 361.859,Z 403.412,A -85,B 0,C 180,E1 -12933.467,E2 -12933.467} C_VEL
LIN {X 0,Y 361.868,Z 403.396,A -85,B 0,C 180,E1 -12937.143,E2 -12937.143} C_VEL
LIN {X 0,Y 361.869,Z 403.403,A -85,B 0,C 180,E1 -12940.721,E2 -12940.721} C_VEL
LIN {X 0,Y 361.899,Z 403.405,A -85,B 0,C 180,E1 -12944.224,E2 -12944.224} C_VEL
LIN {X 0,Y 362.002,Z 403.387,A -85,B 0,C 180,E1 -12946.528,E2 -12946.528} C_VEL
LIN {X 0,Y 361.998,Z 403.381,A -85,B 0,C 180,E1 -12949.937,E2 -12949.937} C_VEL
LIN {X 0,Y 362.122,Z 403.374,A -85,B 0,C 180,E1 -12953.313,E2 -12953.313} C_VEL
LIN {X 0,Y 362.267,Z 403.355,A -85,B 0,C 180,E1 -12957.776,E2 -12957.776} C_VEL
LIN {X 0,Y 362.177,Z 403.36,A -85,B 0,C 180,E1 -12961.112,E2 -12961.112} C_VEL
LIN {X 0,Y 362.262,Z 403.337,A -85,B 0,C 180,E1 -12962.224,E2 -12962.224} C_VEL
LIN {X 0,Y 362.125,Z 403.374,A -85,B 0,C 180,E1 -12966.687,E2 -12966.687} C_VEL
LIN {X 0,Y 361.998,Z 403.373,A -85,B 0,C 180,E1 -12970.063,E2 -12970.063} C_VEL
LIN {X 0,Y 361.983,Z 403.393,A -85,B 0,C 180,E1 -12973.887,E2 -12973.887} C_VEL
LIN {X 0,Y 361.879,Z 403.398,A -85,B 0,C 180,E1 -12978.103,E2 -12978.103} C_VEL
LIN {X 0,Y 361.855,Z 403.402,A -85,B 0,C 180,E1 -12981.655,E2 -12981.655} C_VEL
LIN {X 0,Y 361.868,Z 403.405,A -85,B 0,C 180,E1 -12985.295,E2 -12985.295} C_VEL
LIN {X 0,Y 361.858,Z 403.393,A -85,B 0,C 180,E1 -12989.073,E2 -12989.073} C_VEL
LIN {X 0,Y 361.85,Z 403.408,A -85,B 0,C 180,E1 -12992.945,E2 -12992.945} C_VEL
LIN {X 0,Y 361.865,Z 403.402,A -85,B 0,C 180,E1 -12995.637,E2 -12995.637} C_VEL
LIN {X 0,Y 361.826,Z 403.399,A -85,B 0,C 180,E1 -12999.017,E2 -12999.017} C_VEL
LIN {X 0,Y 361.83,Z 403.381,A -85,B 0,C 180,E1 -13002.83,E2 -13002.83} C_VEL
LIN {X 0,Y 361.815,Z 403.415,A -85,B 0,C 180,E1 -13005.947,E2 -13005.947} C_VEL
LIN {X 0,Y 361.811,Z 403.38,A -85,B 0,C 180,E1 -13009.249,E2 -13009.249} C_VEL
LIN {X 0,Y 361.861,Z 403.411,A -85,B 0,C 180,E1 -13012.981,E2 -13012.981} C_VEL
LIN {X 0,Y 361.933,Z 403.627,A -85,B 0,C 180,E1 -13015.496,E2 -13015.496} C_VEL
LIN {X 0,Y 366.566,Z 424.443,A -85,B 0,C 180,E1 -13019.629,E2 -13019.629} C_VEL
LIN {X 0,Y 367.548,Z 429.014,A -85,B 0,C 180,E1 -13020.503,E2 -13020.503} C_VEL
LIN {X 0,Y 366.203,Z 444.354,A -85,B 0,C 180,E1 -13023.192,E2 -13023.192} C_VEL
LIN {X 0,Y 364.511,Z 464.552,A -85,B 0,C 180,E1 -13026.68,E2 -13026.68} C_VEL
LIN {X 0,Y 366.136,Z 488.732,A -85,B 0,C 180,E1 -13028.153,E2 -13028.153} C_VEL
LIN {X 0,Y 369.614,Z 519.744,A -85,B 0,C 180,E1 -13029.001,E2 -13029.001} C_VEL
LIN {X 0,Y 369.636,Z 533.944,A -85,B 0,C 180,E1 -13029.29,E2 -13029.29} C_VEL
LIN {X 0,Y 368.484,Z 606.502,A -85,B 0,C 180,E1 -13030.719,E2 -13030.719} C_VEL
LIN {X 0,Y 367.789,Z 619.623,A -85,B 0,C 180,E1 -13031.188,E2 -13031.188} C_VEL
LIN {X 0,Y 367.091,Z 632.216,A -85,B 0,C 180,E1 -13031.874,E2 -13031.874} C_VEL
LIN {X 0,Y 366.2,Z 643.421,A -85,B 0,C 180,E1 -13032.694,E2 -13032.694} C_VEL
LIN {X 0,Y 365.106,Z 654.952,A -85,B 0,C 180,E1 -13033.792,E2 -13033.792} C_VEL
LIN {X 0,Y 364.182,Z 664.61,A -85,B 0,C 180,E1 -13034.947,E2 -13034.947} C_VEL
LIN {X 0,Y 363.269,Z 673.768,A -85,B 0,C 180,E1 -13036.291,E2 -13036.291} C_VEL
LIN {X 0,Y 362.385,Z 681.538,A -85,B 0,C 180,E1 -13037.682,E2 -13037.682} C_VEL
LIN {X 0,Y 361.62,Z 689.101,A -85,B 0,C 180,E1 -13039.36,E2 -13039.36} C_VEL
LIN {X 0,Y 361.077,Z 695.17,A -85,B 0,C 180,E1 -13041.042,E2 -13041.042} C_VEL
LIN {X 0,Y 360.691,Z 699.96,A -85,B 0,C 180,E1 -13042.724,E2 -13042.724} C_VEL
LIN {X 0,Y 360.498,Z 703.615,A -85,B 0,C 180,E1 -13044.406,E2 -13044.406} C_VEL
LIN {X 0,Y 360.461,Z 705.498,A -85,B 0,C 180,E1 -13045.527,E2 -13045.527} C_VEL
LIN {X 0,Y 360.363,Z 706.918,A -85,B 0,C 180,E1 -13046.646,E2 -13046.646} C_VEL
LIN {X 0,Y 360.34,Z 708.531,A -85,B 0,C 180,E1 -13048.882,E2 -13048.882} C_VEL
LIN {X 0,Y 360.38,Z 708.75,A -85,B 0,C 180,E1 -13050,E2 -13050} C_VEL
LIN {X 0,Y 360.388,Z 708.528,A -85,B 0,C 180,E1 -13051.117,E2 -13051.117} C_VEL
LIN {X 0,Y 360.37,Z 706.909,A -85,B 0,C 180,E1 -13053.354,E2 -13053.354} C_VEL
LIN {X 0,Y 360.47,Z 705.484,A -85,B 0,C 180,E1 -13054.473,E2 -13054.473} C_VEL
LIN {X 0,Y 360.582,Z 702.274,A -85,B 0,C 180,E1 -13056.265,E2 -13056.265} C_VEL
LIN {X 0,Y 360.785,Z 698.488,A -85,B 0,C 180,E1 -13057.837,E2 -13057.837} C_VEL
LIN {X 0,Y 361.334,Z 692.272,A -85,B 0,C 180,E1 -13059.799,E2 -13059.799} C_VEL
LIN {X 0,Y 361.983,Z 685.486,A -85,B 0,C 180,E1 -13061.479,E2 -13061.479} C_VEL
LIN {X 0,Y 362.75,Z 678.537,A -85,B 0,C 180,E1 -13062.874,E2 -13062.874} C_VEL
LIN {X 0,Y 363.628,Z 670.135,A -85,B 0,C 180,E1 -13064.266,E2 -13064.266} C_VEL
LIN {X 0,Y 364.632,Z 659.729,A -85,B 0,C 180,E1 -13065.655,E2 -13065.655} C_VEL
LIN {X 0,Y 365.613,Z 649.412,A -85,B 0,C 180,E1 -13066.758,E2 -13066.758} C_VEL
LIN {X 0,Y 366.6,Z 638.041,A -85,B 0,C 180,E1 -13067.718,E2 -13067.718} C_VEL
LIN {X 0,Y 367.483,Z 624.961,A -85,B 0,C 180,E1 -13068.539,E2 -13068.539} C_VEL
LIN {X 0,Y 368.194,Z 612.628,A -85,B 0,C 180,E1 -13069.079,E2 -13069.079} C_VEL
LIN {X 0,Y 368.545,Z 600.723,A -85,B 0,C 180,E1 -13069.422,E2 -13069.422} C_VEL
LIN {X 0,Y 369.972,Z 586.214,A -85,B 0,C 180,E1 -13070.139,E2 -13070.139} C_VEL
LIN {X 0,Y 370.789,Z 571.949,A -85,B 0,C 180,E1 -13070.636,E2 -13070.636} C_VEL
LIN {X 0,Y 372.903,Z 522.312,A -85,B 0,C 180,E1 -13072.047,E2 -13072.047} C_VEL
LIN {X 0,Y 371.672,Z 499.369,A -85,B 0,C 180,E1 -13072.959,E2 -13072.959} C_VEL
LIN {X 0,Y 369.403,Z 480.856,A -85,B 0,C 180,E1 -13073.871,E2 -13073.871} C_VEL
LIN {X 0,Y 366.261,Z 462.358,A -85,B 0,C 180,E1 -13074.97,E2 -13074.97} C_VEL
LIN {X 0,Y 368.219,Z 447.314,A -85,B 0,C 180,E1 -13077.88,E2 -13077.88} C_VEL
LIN {X 0,Y 370.087,Z 435.932,A -85,B 0,C 180,E1 -13080.214,E2 -13080.214} C_VEL
LIN {X 0,Y 369.368,Z 430.6,A -85,B 0,C 180,E1 -13081.553,E2 -13081.553} C_VEL
LIN {X 0,Y 367.716,Z 423.07,A -85,B 0,C 180,E1 -13083.66,E2 -13083.66} C_VEL
LIN {X 0,Y 365.615,Z 415.344,A -85,B 0,C 180,E1 -13086.163,E2 -13086.163} C_VEL
LIN {X 0,Y 363.661,Z 409.083,A -85,B 0,C 180,E1 -13088.554,E2 -13088.554} C_VEL
LIN {X 0,Y 361.813,Z 403.535,A -85,B 0,C 180,E1 -13091.164,E2 -13091.164} C_VEL
LIN {X 0,Y 361.812,Z 403.418,A -85,B 0,C 180,E1 -13094.369,E2 -13094.369} C_VEL
LIN {X 0,Y 361.826,Z 403.417,A -85,B 0,C 180,E1 -13097.57,E2 -13097.57} C_VEL
LIN {X 0,Y 361.843,Z 403.411,A -85,B 0,C 180,E1 -13101.572,E2 -13101.572} C_VEL
LIN {X 0,Y 361.875,Z 403.41,A -85,B 0,C 180,E1 -13104.655,E2 -13104.655} C_VEL
LIN {X 0,Y 361.839,Z 403.415,A -85,B 0,C 180,E1 -13108.371,E2 -13108.371} C_VEL
LIN {X 0,Y 361.867,Z 403.407,A -85,B 0,C 180,E1 -13110.952,E2 -13110.952} C_VEL
LIN {X 0,Y 361.908,Z 403.534,A -85,B 0,C 180,E1 -13114.554,E2 -13114.554} C_VEL
LIN {X 0,Y 362.095,Z 404.471,A -85,B 0,C 180,E1 -13114.812,E2 -13114.812} C_VEL
LIN {X 0,Y 363.654,Z 407.275,A -85,B 0,C 180,E1 -13115.194,E2 -13115.194} C_VEL
LIN {X 0,Y 364.647,Z 408.572,A -85,B 0,C 180,E1 -13115.401,E2 -13115.401} C_VEL
LIN {X 0,Y 366.592,Z 411.806,A -85,B 0,C 180,E1 -13115.816,E2 -13115.816} C_VEL
LIN {X 0,Y 372.886,Z 423.061,A -85,B 0,C 180,E1 -13117.093,E2 -13117.093} C_VEL
LIN {X 0,Y 376.253,Z 429.987,A -85,B 0,C 180,E1 -13117.758,E2 -13117.758} C_VEL
LIN {X 0,Y 373.47,Z 482.433,A -85,B 0,C 180,E1 -13119.339,E2 -13119.339} C_VEL
LIN {X 0,Y 373.136,Z 499.854,A -85,B 0,C 180,E1 -13119.967,E2 -13119.967} C_VEL
LIN {X 0,Y 372.577,Z 513.697,A -85,B 0,C 180,E1 -13120.714,E2 -13120.714} C_VEL
LIN {X 0,Y 371.837,Z 525.993,A -85,B 0,C 180,E1 -13121.616,E2 -13121.616} C_VEL
LIN {X 0,Y 370.757,Z 538.176,A -85,B 0,C 180,E1 -13122.771,E2 -13122.771} C_VEL
LIN {X 0,Y 369.74,Z 547.385,A -85,B 0,C 180,E1 -13123.86,E2 -13123.86} C_VEL
LIN {X 0,Y 368.749,Z 555.961,A -85,B 0,C 180,E1 -13125.09,E2 -13125.09} C_VEL
LIN {X 0,Y 367.511,Z 565.209,A -85,B 0,C 180,E1 -13126.734,E2 -13126.734} C_VEL
LIN {X 0,Y 366.601,Z 571.112,A -85,B 0,C 180,E1 -13128.027,E2 -13128.027} C_VEL
LIN {X 0,Y 365.668,Z 576.572,A -85,B 0,C 180,E1 -13129.48,E2 -13129.48} C_VEL
LIN {X 0,Y 364.733,Z 581.511,A -85,B 0,C 180,E1 -13131.132,E2 -13131.132} C_VEL
LIN {X 0,Y 364.053,Z 585.251,A -85,B 0,C 180,E1 -13132.791,E2 -13132.791} C_VEL
LIN {X 0,Y 363.336,Z 587.92,A -85,B 0,C 180,E1 -13134.45,E2 -13134.45} C_VEL
LIN {X 0,Y 363.122,Z 589.082,A -85,B 0,C 180,E1 -13135.56,E2 -13135.56} C_VEL
LIN {X 0,Y 362.837,Z 589.822,A -85,B 0,C 180,E1 -13136.669,E2 -13136.669} C_VEL
LIN {X 0,Y 362.601,Z 590.15,A -85,B 0,C 180,E1 -13137.778,E2 -13137.778} C_VEL
LIN {X 0,Y 362.313,Z 590.06,A -85,B 0,C 180,E1 -13138.889,E2 -13138.889} C_VEL
LIN {X 0,Y 362.09,Z 589.504,A -85,B 0,C 180,E1 -13140,E2 -13140} C_VEL
LIN {X 0,Y 362.088,Z 588.516,A -85,B 0,C 180,E1 -13141.112,E2 -13141.112} C_VEL
LIN {X 0,Y 362.022,Z 587.123,A -85,B 0,C 180,E1 -13142.225,E2 -13142.225} C_VEL
LIN {X 0,Y 362.04,Z 584.154,A -85,B 0,C 180,E1 -13143.896,E2 -13143.896} C_VEL
LIN {X 0,Y 362.221,Z 580.096,A -85,B 0,C 180,E1 -13145.567,E2 -13145.567} C_VEL
LIN {X 0,Y 362.557,Z 573.843,A -85,B 0,C 180,E1 -13147.519,E2 -13147.519} C_VEL
LIN {X 0,Y 362.934,Z 567.153,A -85,B 0,C 180,E1 -13149.164,E2 -13149.164} C_VEL
LIN {X 0,Y 363.369,Z 558.515,A -85,B 0,C 180,E1 -13150.87,E2 -13150.87} C_VEL
LIN {X 0,Y 363.862,Z 549.839,A -85,B 0,C 180,E1 -13152.267,E2 -13152.267} C_VEL
LIN {X 0,Y 364.383,Z 539.25,A -85,B 0,C 180,E1 -13153.667,E2 -13153.667} C_VEL
LIN {X 0,Y 365.03,Z 527.323,A -85,B 0,C 180,E1 -13154.923,E2 -13154.923} C_VEL
LIN {X 0,Y 365.427,Z 515.407,A -85,B 0,C 180,E1 -13155.926,E2 -13155.926} C_VEL
LIN {X 0,Y 365.831,Z 501.342,A -85,B 0,C 180,E1 -13156.82,E2 -13156.82} C_VEL
LIN {X 0,Y 366.105,Z 488.166,A -85,B 0,C 180,E1 -13157.419,E2 -13157.419} C_VEL
LIN {X 0,Y 366.255,Z 467.711,A -85,B 0,C 180,E1 -13157.999,E2 -13157.999} C_VEL
LIN {X 0,Y 367.212,Z 420.286,A -85,B 0,C 180,E1 -13159.209,E2 -13159.209} C_VEL
LIN {X 0,Y 362.088,Z 404.284,A -85,B 0,C 180,E1 -13159.857,E2 -13159.857} C_VEL
LIN {X 0,Y 361.912,Z 403.47,A -85,B 0,C 180,E1 -13160.079,E2 -13160.079} C_VEL
LIN {X 0,Y 361.907,Z 403.404,A -85,B 0,C 180,E1 -13164.067,E2 -13164.067} C_VEL
LIN {X 0,Y 361.851,Z 403.402,A -85,B 0,C 180,E1 -13167.784,E2 -13167.784} C_VEL
LIN {X 0,Y 361.848,Z 403.412,A -85,B 0,C 180,E1 -13171.285,E2 -13171.285} C_VEL
LIN {X 0,Y 361.856,Z 403.397,A -85,B 0,C 180,E1 -13174.28,E2 -13174.28} C_VEL
LIN {X 0,Y 361.865,Z 403.404,A -85,B 0,C 180,E1 -13177.223,E2 -13177.223} C_VEL
LIN {X 0,Y 361.836,Z 403.413,A -85,B 0,C 180,E1 -13180.755,E2 -13180.755} C_VEL
LIN {X 0,Y 361.819,Z 403.415,A -85,B 0,C 180,E1 -13184.369,E2 -13184.369} C_VEL
LIN {X 0,Y 361.837,Z 403.409,A -85,B 0,C 180,E1 -13187.568,E2 -13187.568} C_VEL
LIN {X 0,Y 361.831,Z 403.394,A -85,B 0,C 180,E1 -13190.981,E2 -13190.981} C_VEL
LIN {X 0,Y 361.923,Z 403.615,A -85,B 0,C 180,E1 -13194.284,E2 -13194.284} C_VEL
LIN {X 0,Y 365.508,Z 416.31,A -85,B 0,C 180,E1 -13196.764,E2 -13196.764} C_VEL
LIN {X 0,Y 369.042,Z 430.712,A -85,B 0,C 180,E1 -13199.391,E2 -13199.391} C_VEL
LIN {X 0,Y 370.014,Z 436.515,A -85,B 0,C 180,E1 -13200.407,E2 -13200.407} C_VEL
LIN {X 0,Y 368.334,Z 459.68,A -85,B 0,C 180,E1 -13203.969,E2 -13203.969} C_VEL
LIN {X 0,Y 366.914,Z 481.663,A -85,B 0,C 180,E1 -13207.225,E2 -13207.225} C_VEL
LIN {X 0,Y 366.629,Z 488.017,A -85,B 0,C 180,E1 -13208.085,E2 -13208.085} C_VEL
LIN {X 0,Y 370.299,Z 513.39,A -85,B 0,C 180,E1 -13208.843,E2 -13208.843} C_VEL
LIN {X 0,Y 369.373,Z 576.651,A -85,B 0,C 180,E1 -13210.081,E2 -13210.081} C_VEL
LIN {X 0,Y 368.886,Z 601.284,A -85,B 0,C 180,E1 -13210.597,E2 -13210.597} C_VEL
LIN {X 0,Y 368.284,Z 613.96,A -85,B 0,C 180,E1 -13211.07,E2 -13211.07} C_VEL
LIN {X 0,Y 367.482,Z 627.364,A -85,B 0,C 180,E1 -13211.822,E2 -13211.822} C_VEL
LIN {X 0,Y 366.483,Z 639.047,A -85,B 0,C 180,E1 -13212.708,E2 -13212.708} C_VEL
LIN {X 0,Y 365.399,Z 650.712,A -85,B 0,C 180,E1 -13213.863,E2 -13213.863} C_VEL
LIN {X 0,Y 364.598,Z 659.671,A -85,B 0,C 180,E1 -13214.971,E2 -13214.971} C_VEL
LIN {X 0,Y 363.582,Z 668.611,A -85,B 0,C 180,E1 -13216.303,E2 -13216.303} C_VEL
LIN {X 0,Y 362.64,Z 676.272,A -85,B 0,C 180,E1 -13217.691,E2 -13217.691} C_VEL
LIN {X 0,Y 361.885,Z 683.739,A -85,B 0,C 180,E1 -13219.368,E2 -13219.368} C_VEL
LIN {X 0,Y 361.232,Z 689.733,A -85,B 0,C 180,E1 -13221.046,E2 -13221.046} C_VEL
LIN {X 0,Y 360.841,Z 694.475,A -85,B 0,C 180,E1 -13222.727,E2 -13222.727} C_VEL
LIN {X 0,Y 360.554,Z 698.105,A -85,B 0,C 180,E1 -13224.407,E2 -13224.407} C_VEL
LIN {X 0,Y 360.449,Z 699.974,A -85,B 0,C 180,E1 -13225.527,E2 -13225.527} C_VEL
LIN {X 0,Y 360.319,Z 701.403,A -85,B 0,C 180,E1 -13226.646,E2 -13226.646} C_VEL
LIN {X 0,Y 360.258,Z 703.021,A -85,B 0,C 180,E1 -13228.882,E2 -13228.882} C_VEL
LIN {X 0,Y 360.275,Z 703.256,A -85,B 0,C 180,E1 -13230,E2 -13230} C_VEL
LIN {X 0,Y 360.258,Z 703.063,A -85,B 0,C 180,E1 -13231.118,E2 -13231.118} C_VEL
LIN {X 0,Y 360.319,Z 701.501,A -85,B 0,C 180,E1 -13233.355,E2 -13233.355} C_VEL
LIN {X 0,Y 360.445,Z 700.127,A -85,B 0,C 180,E1 -13234.473,E2 -13234.473} C_VEL
LIN {X 0,Y 360.6,Z 696.956,A -85,B 0,C 180,E1 -13236.289,E2 -13236.289} C_VEL
LIN {X 0,Y 361.015,Z 691.743,A -85,B 0,C 180,E1 -13238.396,E2 -13238.396} C_VEL
LIN {X 0,Y 361.136,Z 690.658,A -85,B 0,C 180,E1 -13238.754,E2 -13238.754} C_VEL
LIN {X 0,Y 360.77,Z 688.041,A -85,B 0,C 180,E1 -13239.593,E2 -13239.593} C_VEL
LIN {X 0,Y 358.411,Z 683.4,A -85,B 0,C 180,E1 -13240.941,E2 -13240.941} C_VEL
LIN {X 0,Y 356.153,Z 678.154,A -85,B 0,C 180,E1 -13242.244,E2 -13242.244} C_VEL
LIN {X 0,Y 355.944,Z 674.557,A -85,B 0,C 180,E1 -13243,E2 -13243} C_VEL
LIN {X 0,Y 357.061,Z 665.806,A -85,B 0,C 180,E1 -13244.534,E2 -13244.534} C_VEL
LIN {X 0,Y 357.934,Z 656.848,A -85,B 0,C 180,E1 -13245.822,E2 -13245.822} C_VEL
LIN {X 0,Y 359.071,Z 645.957,A -85,B 0,C 180,E1 -13247.073,E2 -13247.073} C_VEL
LIN {X 0,Y 360.128,Z 635.271,A -85,B 0,C 180,E1 -13248.048,E2 -13248.048} C_VEL
LIN {X 0,Y 361.067,Z 623.546,A -85,B 0,C 180,E1 -13248.881,E2 -13248.881} C_VEL
LIN {X 0,Y 361.805,Z 611.53,A -85,B 0,C 180,E1 -13249.504,E2 -13249.504} C_VEL
LIN {X 0,Y 362.355,Z 598.402,A -85,B 0,C 180,E1 -13249.953,E2 -13249.953} C_VEL
LIN {X 0,Y 363.768,Z 514.405,A -85,B 0,C 180,E1 -13251.638,E2 -13251.638} C_VEL
LIN {X 0,Y 359.954,Z 487.728,A -85,B 0,C 180,E1 -13252.472,E2 -13252.472} C_VEL
LIN {X 0,Y 361.094,Z 468.023,A -85,B 0,C 180,E1 -13255.353,E2 -13255.353} C_VEL
LIN {X 0,Y 362.884,Z 444.587,A -85,B 0,C 180,E1 -13258.959,E2 -13258.959} C_VEL
LIN {X 0,Y 363.342,Z 438.418,A -85,B 0,C 180,E1 -13259.939,E2 -13259.939} C_VEL
LIN {X 0,Y 361.961,Z 430.701,A -85,B 0,C 180,E1 -13261.314,E2 -13261.314} C_VEL
LIN {X 0,Y 358.085,Z 415.382,A -85,B 0,C 180,E1 -13264.198,E2 -13264.198} C_VEL
LIN {X 0,Y 354.856,Z 404.472,A -85,B 0,C 180,E1 -13266.382,E2 -13266.382} C_VEL
LIN {X 0,Y 354.77,Z 404.281,A -85,B 0,C 180,E1 -13269.413,E2 -13269.413} C_VEL
LIN {X 0,Y 354.786,Z 404.291,A -85,B 0,C 180,E1 -13272.867,E2 -13272.867} C_VEL
LIN {X 0,Y 354.767,Z 404.28,A -85,B 0,C 180,E1 -13276.103,E2 -13276.103} C_VEL
LIN {X 0,Y 354.768,Z 404.289,A -85,B 0,C 180,E1 -13279.176,E2 -13279.176} C_VEL
LIN {X 0,Y 354.802,Z 404.28,A -85,B 0,C 180,E1 -13282.405,E2 -13282.405} C_VEL
LIN {X 0,Y 354.811,Z 404.288,A -85,B 0,C 180,E1 -13284.94,E2 -13284.94} C_VEL
LIN {X 0,Y 354.797,Z 404.29,A -85,B 0,C 180,E1 -13288.405,E2 -13288.405} C_VEL
LIN {X 0,Y 354.8,Z 404.279,A -85,B 0,C 180,E1 -13291.614,E2 -13291.614} C_VEL
LIN {X 0,Y 354.837,Z 404.273,A -85,B 0,C 180,E1 -13295.657,E2 -13295.657} C_VEL
LIN {X 0,Y 354.829,Z 404.286,A -85,B 0,C 180,E1 -13299.113,E2 -13299.113} C_VEL
LIN {X 0,Y 354.855,Z 404.266,A -85,B 0,C 180,E1 -13302.718,E2 -13302.718} C_VEL
LIN {X 0,Y 354.943,Z 404.268,A -85,B 0,C 180,E1 -13306.255,E2 -13306.255} C_VEL
LIN {X 0,Y 354.954,Z 404.254,A -85,B 0,C 180,E1 -13309.735,E2 -13309.735} C_VEL
LIN {X 0,Y 355.089,Z 404.251,A -85,B 0,C 180,E1 -13313.18,E2 -13313.18} C_VEL
LIN {X 0,Y 355.229,Z 404.231,A -85,B 0,C 180,E1 -13317.732,E2 -13317.732} C_VEL
LIN {X 0,Y 355.148,Z 404.235,A -85,B 0,C 180,E1 -13321.134,E2 -13321.134} C_VEL
LIN {X 0,Y 355.223,Z 404.213,A -85,B 0,C 180,E1 -13322.268,E2 -13322.268} C_VEL
LIN {X 0,Y 355.091,Z 404.251,A -85,B 0,C 180,E1 -13326.82,E2 -13326.82} C_VEL
LIN {X 0,Y 354.954,Z 404.251,A -85,B 0,C 180,E1 -13330.265,E2 -13330.265} C_VEL
LIN {X 0,Y 354.921,Z 404.271,A -85,B 0,C 180,E1 -13334.002,E2 -13334.002} C_VEL
LIN {X 0,Y 354.837,Z 404.274,A -85,B 0,C 180,E1 -13338.064,E2 -13338.064} C_VEL
LIN {X 0,Y 354.808,Z 404.273,A -85,B 0,C 180,E1 -13342.108,E2 -13342.108} C_VEL
LIN {X 0,Y 354.804,Z 404.29,A -85,B 0,C 180,E1 -13345.835,E2 -13345.835} C_VEL
LIN {X 0,Y 354.799,Z 404.275,A -85,B 0,C 180,E1 -13349.684,E2 -13349.684} C_VEL
LIN {X 0,Y 354.789,Z 404.289,A -85,B 0,C 180,E1 -13352.333,E2 -13352.333} C_VEL
LIN {X 0,Y 354.82,Z 404.28,A -85,B 0,C 180,E1 -13355.698,E2 -13355.698} C_VEL
LIN {X 0,Y 354.77,Z 404.267,A -85,B 0,C 180,E1 -13359.412,E2 -13359.412} C_VEL
LIN {X 0,Y 354.782,Z 404.258,A -85,B 0,C 180,E1 -13362.866,E2 -13362.866} C_VEL
LIN {X 0,Y 354.764,Z 404.291,A -85,B 0,C 180,E1 -13366.103,E2 -13366.103} C_VEL
LIN {X 0,Y 354.763,Z 404.256,A -85,B 0,C 180,E1 -13369.175,E2 -13369.175} C_VEL
LIN {X 0,Y 354.799,Z 404.292,A -85,B 0,C 180,E1 -13372.404,E2 -13372.404} C_VEL
LIN {X 0,Y 354.895,Z 404.442,A -85,B 0,C 180,E1 -13375.217,E2 -13375.217} C_VEL
LIN {X 0,Y 359.388,Z 424.908,A -85,B 0,C 180,E1 -13379.366,E2 -13379.366} C_VEL
LIN {X 0,Y 360.565,Z 430.851,A -85,B 0,C 180,E1 -13380.517,E2 -13380.517} C_VEL
LIN {X 0,Y 358.944,Z 447.826,A -85,B 0,C 180,E1 -13383.549,E2 -13383.549} C_VEL
LIN {X 0,Y 357.759,Z 461.787,A -85,B 0,C 180,E1 -13386.021,E2 -13386.021} C_VEL
LIN {X 0,Y 358.064,Z 467.842,A -85,B 0,C 180,E1 -13386.427,E2 -13386.427} C_VEL
